// TwinCAT 3 PLC project PLC
// ProgramVersion: 3.1.4024.0
// libraries:
//   SPT Base Types, * (Beckhoff Automation LLC)
//   SPT Components, * (Beckhoff Automation LLC)
//   SPT Event Logger, * (Beckhoff Automation LLC)
//   SPT Motion Control, * (Beckhoff Automation LLC)
//   SPT Utilities, * (Beckhoff Automation LLC)
//   Tc2_MC2, * (Beckhoff Automation GmbH)
//   Tc2_MC2_Drive, * (Beckhoff Automation GmbH)
//   Tc2_NCI, * (Beckhoff Automation GmbH)
//   Tc2_PlcInterpolation, * (Beckhoff Automation GmbH)
//   Tc2_Standard, * (Beckhoff Automation GmbH)
//   Tc2_System, * (Beckhoff Automation GmbH)
//   Tc2_Utilities, * (Beckhoff Automation GmbH)
//   Tc3_EventLogger, * (Beckhoff Automation GmbH)
//   Tc3_Module, * (Beckhoff Automation GmbH)
//   Tc3_PackML_V2, * (Beckhoff Automation GmbH)
//   TcUnit, * (www.tcunit.org)
//   VisuDialogs, * (System)
// project tree:
//   DUTs/ ST_Recipe_Limits.TcDUT, ST_LimitInfo.TcDUT, E_CutDirection.TcDUT, E_PMLStateForHMI.TcTLEO, ST_Machine_HMI.TcDUT, ST_Machine_Status.TcDUT
//   GVLs/ GVL_HMI.TcGVL, GVL_Safety.TcGVL, IO.TcGVL
//   / PlcTask.TcTTO, SafetyTask.TcTTO, Visualization Manager.TcVMO (not stored), VISU_TASK.TcTTO
//   POUs/Builder/ E_ExecutionRoute.TcDUT, I_GeometryWriter.TcIO, FB_RecipeBase.TcPOU, FB_RecipeFactory.TcPOU, I_RecipeBuilder.TcIO, ST_CutSegment.TcDUT, ST_PointXY.TcDUT (not stored), ST_RecipeBuilder_Config.TcDUT, ST_RecipeBuilder_HMI.TcDUT
//   POUs/Builder/Recipes/ FB_FeedMeina2_1000x1000_Circles.TcPOU, FB_FeedMeina2_2000x500.TcPOU, FB_FeedMeina2_750x750.TcPOU, FB_FeedMeina2_750x750_Circles.TcPOU, FB_FeedMeina2_1000x1000.TcPOU, FB_FeedMeina2_500x500.TcPOU, FB_FeedMeina2_500x500_Circles.TcPOU, FB_FeedRoundedRectangle.TcPOU, FB_FeedCircle.TcPOU, FB_FeedMeina2_2000x1000.TcPOU, FB_FeedMeina2_Samples.TcPOU, FB_PTPArona.TcPOU, FB_NCICircle.TcPOU, FB_PTPRectangle.TcPOU, FB_PTPBorgoFlaps.TcPOU, FB_PTPBorgoWings.TcPOU
//   POUs/Components/ FB_Cylinder.TcPOU, I_Cylinder.TcIO, FB_NciChannel.TcPOU, FB_NciChannelTangential.TcPOU, ST_Cylinder_Command.TcDUT, ST_Cylinder_Config.TcDUT, ST_Cylinder_HMI.TcDUT, ST_Cylinder_Status.TcDUT
//   POUs/Components/I_Channel/ ST_NciAxisIds.TcDUT, I_NciChannelBase.TcIO, I_NciChannel_FeedTable.TcIO, I_NciChannel_GCode.TcIO
//   POUs/Executor/ FB_Exec_Pneumatic_PTP.TcPOU, FB_Exec_Drill_PTP.TcPOU, FB_Exec_Tangential_FeedTable.TcPOU, FB_Exec_Spindle_PTP.TcPOU, I_BB8Specification.TcIO, FB_ExecutorBase.TcPOU, I_MachiningExecutor.TcIO, FB_Exec_Spindle_GCodeXYZ.TcPOU
//   POUs/GantryXYZ/ E_MachineProfile.TcDUT, E_RecipeID.TcDUT, ST_AxisProfile.TcDUT, ST_GantryXYZ_Limits.TcDUT, FB_GantryXYZ.TcPOU, I_GantryConfigProvider.TcIO, ST_GantryXYZ_Command.TcDUT, ST_GantryXYZ_Config.TcDUT, ST_GantryXYZ_HMI.TcDUT, ST_GantryXYZ_Status.TcDUT (not stored)
//   POUs/GantryXYZ/HomingStrategies/ FB_Homing_Base.TcPOU, FB_Homing_CustomPLC.TcPOU, FB_Homing_Direct.TcPOU, FB_Homing_StandardNC.TcPOU, I_HomingStrategy.TcIO
//   POUs/ FB_Machine.TcPOU, FB_PersistentDataManager.TcPOU, GlobalTextList.TcGTLO, MAIN.TcPOU, SAFETY.TcPOU, TESTS.TcPOU
//   POUs/TESTS/ FB_Cylinder_Test.TcPOU, FB_ExecutorNCITable_Test.TcPOU, FB_ExecutorGCode_Test.TcPOU, FB_FeedBuilderRoundedRect_Test.TcPOU, FB_NciChannelTangential_Test.TcPOU, FB_NciChannel_Test.TcPOU, FB_GantryXYZ_Test.TcPOU, FB_ExecutorCut_Test.TcPOU, FB_ExecutorGrooveXY_Test.TcPOU, FB_RecipeBuilder_Test.TcPOU, FB_RecipeFactory_Test.TcPOU, FB_Exec_Drill_PTP_Test.TcPOU
//   POUs/TESTS/Mocks/ FB_MockAxis.TcPOU, FB_MockRecipe_Drill.TcPOU, FB_MockGeometryWriter.TcPOU, FB_MockNciChannelFeedTable.TcPOU, FB_MockNciChannel.TcPOU, FB_MockCylinder.TcPOU, FB_MockConfigProvider.TcPOU
//   VISUs/Modes/ProductionMode/ V_Builders.TcVIS, V_Meina2_Samples.TcVIS, V_ProductionArona.TcVIS, V_ProductionFeedCircle.TcVIS, V_ProductionMeina2_5Squares.TcVIS, V_ProductionMeina2_5Circles.TcVIS, V_ProductionMeina2_3Squares.TcVIS, V_ProductionMeina2_3Circles.TcVIS, V_ProductionMeina2_2Squares.TcVIS, V_ProductionMeina2_2Circles.TcVIS, V_ProductionMeina2_2Rectangles.TcVIS, V_ProductionRoundRectangle.TcVIS, V_ProductionRectangle.TcVIS, V_ProductionNCICircle.TcVIS, V_ProductionBorgoFlaps.TcVIS, V_ProductionBorgoWings.TcVIS, V_Meina2_2000x1000.TcVIS, V_ProductionWelcome.TcVIS
//   VISUs/Modes/ V_MaintenanceMode.TcVIS, V_ManualMode.TcVIS, V_ProductionMode.TcVIS
//   VISUs/ V_InfoMenu.TcVIS, V_MainMenu.TcVIS, V_Main.TcVIS
// real-time tasks:
//   TASK PlcTask: cycle T#10ms, priority 20, ADS port 350
//   TASK SafetyTask: cycle T#10ms, priority 21, ADS port 351
//   TASK VISU_TASK: cycle T#200000us, priority 30, ADS port 352
// motion (NC):
//   TASK NC-Task 1 SAF: cycle T#2ms, priority 4, ADS port 501
//   TASK NC-Task 1 SVB: cycle T#10ms, priority 8, ADS port 511
//   AXIS Test Axis X (id 5)
//     OtherSettings: AllowMotionCmdToSlave=true
//     encoder EncType=1
//       Inc: RefSoftSyncMask=#x0000ffff
//     drive DrvType=5
//       Analog: TorqueSetpointScale=10, ScaleFactorActTorque=0.1
//       TimeComp: TaskDelayCycles=1
//     controller CtrType=1
//       CtrPara: PriorControlFactor=1
//         Observer: BandWidth=20
//   AXIS Test Axis Y (id 6)
//     OtherSettings: AllowMotionCmdToSlave=true
//     encoder EncType=1
//     drive DrvType=5
//       Analog: TorqueSetpointScale=10, ScaleFactorActTorque=0.1
//       TimeComp: TaskDelayCycles=1
//     controller CtrType=1
//       CtrPara: PriorControlFactor=1
//         Observer: BandWidth=20
//   AXIS Test Axis Z (id 7)
//     OtherSettings: AllowMotionCmdToSlave=true
//     encoder EncType=1
//     drive DrvType=5
//       Analog: TorqueSetpointScale=10, ScaleFactorActTorque=0.1
//       TimeComp: TaskDelayCycles=1
//     controller CtrType=1
//       CtrPara: PriorControlFactor=1
//         Observer: BandWidth=20
//   AXIS Test Axis Q (id 8)
//     OtherSettings: AllowMotionCmdToSlave=true
//     encoder EncType=1
//     drive DrvType=5
//       Analog: TorqueSetpointScale=10, ScaleFactorActTorque=0.1
//       TimeComp: TaskDelayCycles=1
//     controller CtrType=1
//       CtrPara: PriorControlFactor=1
//         Observer: BandWidth=20
//   AXIS Axis Q (id 1)
//     General: UnitName=°
//     Dynamic: Acceleration=15000, Deceleration=15000, Jerk=45000
//     Velo: RefSearch=720, RefSync=90, SlowManual=30, FastManual=180, Fast=10738.39, Maximum=10738.4
//     TargetPosControl: Range=0.1
//     BacklashCompensation: Range=0.2
//     OtherSettings: AllowMotionCmdToSlave=true, PulseDistancePos=9, PulseDistanceNeg=9
//     encoder EncType=19
//       EncPara: ScaleFactorNumerator=360, ScaleFactorDenominator=3145728, MaxCount=#xffffffff
//         SoftEndMinControl: Range=-300
//         SoftEndMaxControl: Range=300
//     drive DrvType=16
//       DrvPara: MaxCount=#xffffffff, DriveControlDWord=#x00020100
//         Analog: VeloReferenz=11812.229, VeloScale=32, TorqueSetpointScale=10, ScaleFactorActTorque=0.1
//         TimeComp: TaskDelayCycles=1
//     controller CtrType=1
//       CtrPara: PriorControlFactor=1
//         PosDiffControl: Range=40
//         Observer: BandWidth=20
//   AXIS Axis Y (id 2)
//     Dynamic: Acceleration=100, Deceleration=100, Jerk=200
//     Velo: RefSearch=50, RefSync=10, SlowManual=5, FastManual=80, Fast=429.536, Maximum=429.536
//     TargetPosControl: Range=0.1
//     BacklashCompensation: Range=0.1
//     OtherSettings: AllowMotionCmdToSlave=true
//     encoder EncType=19
//       EncPara: ScaleFactorNumerator=4.8, ScaleFactorDenominator=1048576, MaxCount=#xffffffff
//         SoftEndMinControl: Enable=true, Range=-3000
//         SoftEndMaxControl: Enable=true, Range=3000
//         Inc: RefSearchInverse=true, RefSyncInverse=false, RefMode=1
//     drive DrvType=16
//       DrvPara: MaxCount=#xffffffff, DriveControlDWord=#x00020100
//         Analog: VeloReferenz=472.4896, VeloScale=32, TorqueSetpointScale=10, ScaleFactorActTorque=0.1
//         TimeComp: TaskDelayCycles=1
//     controller CtrType=1
//       CtrPara: PriorControlFactor=1
//         Observer: BandWidth=20
//   AXIS Axis Z (id 9)
//     Dynamic: AccelerationMaximum=1200, DecelerationMaximum=1200, Acceleration=20, Deceleration=20, Jerk=80
//     Velo: RefSearch=5, RefSync=2, SlowManual=5, FastManual=10, Maximum=20
//     TargetPosControl: Range=0.1
//     BacklashCompensation: Range=0.1
//     OtherSettings: AllowMotionCmdToSlave=true
//     encoder EncType=4
//       EncPara: ScaleFactorNumerator=2, ScaleFactorDenominator=12800, Inverse=true, MaxCount=#xffffffff
//         Inc: RefPosition=31, RefMode=1
//     drive DrvType=24
//       DrvPara: Inverse=true
//         Analog: VeloReferenz=20, TorqueSetpointScale=10, ScaleFactorActTorque=0.1
//         TimeComp: TaskDelayCycles=1
//     controller CtrType=1
//       CtrPara: PriorControlFactor=1
//         PosDiffControl: Range=2
//         Observer: BandWidth=20
//   AXIS Axis X (id 3)
//     Dynamic: Acceleration=100, Deceleration=100, Jerk=200
//     Velo: RefSearch=50, RefSync=10, SlowManual=5, FastManual=80, Fast=536.92, Maximum=536.92
//     TargetPosControl: Range=0.1
//     BacklashCompensation: Range=0.067
//     OtherSettings: AllowMotionCmdToSlave=true
//     encoder EncType=19
//       EncPara: ScaleFactorNumerator=6, ScaleFactorDenominator=1048576, MaxCount=#xffffffff
//         SoftEndMinControl: Enable=true, Range=-2000
//         SoftEndMaxControl: Enable=true, Range=2000
//         Inc: RefSearchInverse=true, RefSyncInverse=false, RefMode=1
//     drive DrvType=16
//       DrvPara: MaxCount=#xffffffff, DriveControlDWord=#x00020100
//         Analog: VeloReferenz=590.612, VeloScale=32, TorqueSetpointScale=10, ScaleFactorActTorque=0.1
//         TimeComp: TaskDelayCycles=1
//     controller CtrType=1
//       CtrPara: PriorControlFactor=1
//         Observer: BandWidth=20
// I/O:
//   DEVICE Device 3 (EtherCAT), AmsNetId 0.0.0.0.4.1
//     Term 1 (EK1100) [EK1100 EtherCAT Coupler (2A E-Bus)]
//       Term 2 (EL1008) [EL1008 8Ch. Dig. Input 24V, 3ms]
//       Term 3 (EL1008) [EL1008 8Ch. Dig. Input 24V, 3ms]
//       Term 4 (EL2008) [EL2008 8Ch. Dig. Output 24V, 0.5A]
//       Term 5 (EL7221-9014) [EL7221-9014 1Ch. MDP742 Servo motor output stage with OCT (50V, 8A RMS) and STO input]
//         startup 32786:19 := 0000 // DRV Brake Settings / Emergency application timeout
//         startup 32784:51 := 0A00 // DRV Amplifier Settings / Stand still window
//         startup 32785:27 := 01150000 // DRV Motor Settings / Motor speed limitation
//         startup 28688:11 := E803 // DRV Outputs / Torque limitation
//         startup 32784:19 := 5300 // DRV Amplifier Settings / Current loop proportional gain
//         startup 32784:18 := 0500 // DRV Amplifier Settings / Current loop integral time
//         startup 32784:21 := 1F010000 // DRV Amplifier Settings / Velocity loop proportional gain
//         startup 32784:20 := 96000000 // DRV Amplifier Settings / Velocity loop integral time
//         startup 32768:1 := 00 // FB Settings / Invert feedback direction
//       Term 6 (EL7221-9014) [EL7221-9014 1Ch. MDP742 Servo motor output stage with OCT (50V, 8A RMS) and STO input]
//         startup 32785:27 := 01150000 // DRV Motor Settings / Motor speed limitation
//         startup 28688:11 := E803 // DRV Outputs / Torque limitation
//         startup 32784:19 := 5300 // DRV Amplifier Settings / Current loop proportional gain
//         startup 32784:18 := 0500 // DRV Amplifier Settings / Current loop integral time
//         startup 32784:21 := E0000000 // DRV Amplifier Settings / Velocity loop proportional gain
//         startup 32784:20 := 96000000 // DRV Amplifier Settings / Velocity loop integral time
//         startup 32768:1 := 00 // FB Settings / Invert feedback direction
//       Term 7 (EL7221-9014) [EL7221-9014 1Ch. MDP742 Servo motor output stage with OCT (50V, 8A RMS) and STO input]
//         startup 32785:27 := 01150000 // DRV Motor Settings / Motor speed limitation
//         startup 28688:11 := E803 // DRV Outputs / Torque limitation
//         startup 32784:19 := 5300 // DRV Amplifier Settings / Current loop proportional gain
//         startup 32784:18 := 0500 // DRV Amplifier Settings / Current loop integral time
//         startup 32784:21 := E0000000 // DRV Amplifier Settings / Velocity loop proportional gain
//         startup 32784:20 := 96000000 // DRV Amplifier Settings / Velocity loop integral time
//         startup 32768:1 := 00 // FB Settings / Invert feedback direction
//       Term 20 (EL7037) [EL7037 1Ch. Stepper motor output stage (24V, 1.5A)]
//       Term 8 (EL6900) [EL6900, TwinSAFE PLC]
//       Term 9 (EL1904) [EL1904, 4 Ch. Safety Input 24V, TwinSAFE]
//         modules: Module 1 (FSOES)
//       Term 10 (EL2904) [EL2904, 4 Ch. Safety Output 24V, 0.5A, TwinSAFE]
//         modules: Module 1 (FSOES), Module 2 (DO)
//       Term 11 (EL2622) [EL2622 2Ch. Relay Output, NO (230V AC / 30V DC)]
//       Term 12 (EL9011) [EL9011 End Terminal]
// variable links:
//   Device 3 (EtherCAT) <-> Device 3 (EtherCAT)/Term 1 (EK1100)/Term 8 (EL6900)
//     Term 1 (EK1100)/Term 10 (EL2904)/Module 1 (FSOES)/RxPDO/FSOE <-> ConnectionInputs/TwinSafeGroup1.Term 10 (EL2904) - Module 1 (FSOES)_3 TxPDO
//     Term 1 (EK1100)/Term 9 (EL1904)/Module 1 (FSOES)/RxPDO/FSOE <-> ConnectionInputs/TwinSafeGroup1.Term 9 (EL1904) - Module 1 (FSOES)_2 TxPDO
//     Term 1 (EK1100)/Term 10 (EL2904)/Module 1 (FSOES)/TxPDO/FSOE <-> ConnectionOutputs/TwinSafeGroup1.Term 10 (EL2904) - Module 1 (FSOES)_3 RxPDO
//     Term 1 (EK1100)/Term 9 (EL1904)/Module 1 (FSOES)/TxPDO/FSOE <-> ConnectionOutputs/TwinSafeGroup1.Term 9 (EL1904) - Module 1 (FSOES)_2 RxPDO
//   NC-Task 1 SAF/Axes/Axis Q <-> Device 3 (EtherCAT)/Term 1 (EK1100)/Term 5 (EL7221-9014)
//     Drive/Inputs/In/nDataIn1 <-> DRV Following error actual value/Following error actual value
//     Drive/Inputs/In/nDataIn3[0] <-> DRV Torque actual value/Torque actual value
//     Drive/Inputs/In/nDcOutputTime <-> InfoData/DcOutputShift
//     Drive/Inputs/In/nState1 <-> DRV Statusword/Statusword
//     Drive/Inputs/In/nState2 <-> DRV Statusword/Statusword @bit 8
//     Drive/Inputs/In/nState4 @bit 1 <-> WcState/InputToggle
//     Drive/Inputs/In/nState4 <-> WcState/WcState
//     Drive/Outputs/Out/nCtrl1 <-> DRV Controlword/Controlword
//     Drive/Outputs/Out/nCtrl2 <-> DRV Controlword/Controlword @bit 8
//     Drive/Outputs/Out/nDataOut1 <-> DRV Target position/Target position
//     Drive/Outputs/Out/nDataOut2 <-> DRV Target velocity/Target velocity
//     Enc/Inputs/In/nDataIn1 <-> FB Position/Position
//     Enc/Inputs/In/nDcInputTime <-> InfoData/DcInputShift
//     Enc/Inputs/In/nState4 @bit 1 <-> WcState/InputToggle
//     Enc/Inputs/In/nState4 <-> WcState/WcState
//   NC-Task 1 SAF/Axes/Axis X <-> Device 3 (EtherCAT)/Term 1 (EK1100)/Term 7 (EL7221-9014)
//     Drive/Inputs/In/nDataIn1 <-> DRV Following error actual value/Following error actual value
//     Drive/Inputs/In/nDataIn3[0] <-> DRV Torque actual value/Torque actual value
//     Drive/Inputs/In/nDcOutputTime <-> InfoData/DcOutputShift
//     Drive/Inputs/In/nState1 <-> DRV Statusword/Statusword
//     Drive/Inputs/In/nState2 <-> DRV Statusword/Statusword @bit 8
//     Drive/Inputs/In/nState4 @bit 1 <-> WcState/InputToggle
//     Drive/Inputs/In/nState4 <-> WcState/WcState
//     Drive/Outputs/Out/nCtrl1 <-> DRV Controlword/Controlword
//     Drive/Outputs/Out/nCtrl2 <-> DRV Controlword/Controlword @bit 8
//     Drive/Outputs/Out/nDataOut1 <-> DRV Target position/Target position
//     Drive/Outputs/Out/nDataOut2 <-> DRV Target velocity/Target velocity
//     Enc/Inputs/In/nDataIn1 <-> FB Position/Position
//     Enc/Inputs/In/nDcInputTime <-> InfoData/DcInputShift
//     Enc/Inputs/In/nState4 @bit 1 <-> WcState/InputToggle
//     Enc/Inputs/In/nState4 <-> WcState/WcState
//   NC-Task 1 SAF/Axes/Axis Y <-> Device 3 (EtherCAT)/Term 1 (EK1100)/Term 6 (EL7221-9014)
//     Drive/Inputs/In/nDataIn1 <-> DRV Following error actual value/Following error actual value
//     Drive/Inputs/In/nDataIn3[0] <-> DRV Torque actual value/Torque actual value
//     Drive/Inputs/In/nDcOutputTime <-> InfoData/DcOutputShift
//     Drive/Inputs/In/nState1 <-> DRV Statusword/Statusword
//     Drive/Inputs/In/nState2 <-> DRV Statusword/Statusword @bit 8
//     Drive/Inputs/In/nState4 @bit 1 <-> WcState/InputToggle
//     Drive/Inputs/In/nState4 <-> WcState/WcState
//     Drive/Outputs/Out/nCtrl1 <-> DRV Controlword/Controlword
//     Drive/Outputs/Out/nCtrl2 <-> DRV Controlword/Controlword @bit 8
//     Drive/Outputs/Out/nDataOut1 <-> DRV Target position/Target position
//     Drive/Outputs/Out/nDataOut2 <-> DRV Target velocity/Target velocity
//     Enc/Inputs/In/nDataIn1 <-> FB Position/Position
//     Enc/Inputs/In/nDcInputTime <-> InfoData/DcInputShift
//     Enc/Inputs/In/nState4 @bit 1 <-> WcState/InputToggle
//     Enc/Inputs/In/nState4 <-> WcState/WcState
//   NC-Task 1 SAF/Axes/Axis Z <-> Device 3 (EtherCAT)/Term 1 (EK1100)/Term 20 (EL7037)
//     Drive/Inputs/In/nState1 @bit 3 <-> STM Status/Error
//     Drive/Inputs/In/nState1 @bit 7 <-> STM Status/Motor stall
//     Drive/Inputs/In/nState1 @bit 5 <-> STM Status/Moving negative
//     Drive/Inputs/In/nState1 @bit 4 <-> STM Status/Moving positive
//     Drive/Inputs/In/nState1 @bit 1 <-> STM Status/Ready
//     Drive/Inputs/In/nState1 <-> STM Status/Ready to enable
//     Drive/Inputs/In/nState1 @bit 6 <-> STM Status/Torque reduced
//     Drive/Inputs/In/nState1 @bit 2 <-> STM Status/Warning
//     Drive/Inputs/In/nState2 @bit 3 <-> STM Status/Digital input 1
//     Drive/Inputs/In/nState2 @bit 4 <-> STM Status/Digital input 2
//     Drive/Inputs/In/nState2 @bit 5 <-> STM Status/Sync error
//     Drive/Inputs/In/nState2 @bit 7 <-> STM Status/TxPDO Toggle
//     Drive/Inputs/In/nState4 @bit 1 <-> WcState/InputToggle
//     Drive/Inputs/In/nState4 <-> WcState/WcState
//     Drive/Outputs/Out/nCtrl1 <-> STM Control/Enable
//     Drive/Outputs/Out/nCtrl1 @bit 2 <-> STM Control/Reduce torque
//     Drive/Outputs/Out/nCtrl1 @bit 1 <-> STM Control/Reset
//     Drive/Outputs/Out/nCtrl2 @bit 3 <-> STM Control/Digital output 1
//     Drive/Outputs/Out/nDataOut1 <-> STM Position/Position
//     Enc/Inputs/In/nDataIn1 <-> ENC Status/Counter value
//     Enc/Inputs/In/nDataIn2 <-> ENC Status/Latch value
//     Enc/Inputs/In/nState1 @bit 4 <-> ENC Status/Counter overflow
//     Enc/Inputs/In/nState1 @bit 3 <-> ENC Status/Counter underflow
//     Enc/Inputs/In/nState1 @bit 7 <-> ENC Status/Extrapolation stall
//     Enc/Inputs/In/nState1 <-> ENC Status/Latch C valid
//     Enc/Inputs/In/nState1 @bit 1 <-> ENC Status/Latch extern valid
//     Enc/Inputs/In/nState1 @bit 2 <-> ENC Status/Set counter done
//     Enc/Inputs/In/nState2 @bit 4 <-> ENC Status/Status of extern latch
//     Enc/Inputs/In/nState2 <-> ENC Status/Status of input A
//     Enc/Inputs/In/nState2 @bit 1 <-> ENC Status/Status of input B
//     Enc/Inputs/In/nState2 @bit 2 <-> ENC Status/Status of input C
//     Enc/Inputs/In/nState2 @bit 5 <-> ENC Status/Sync error
//     Enc/Inputs/In/nState2 @bit 7 <-> ENC Status/TxPDO Toggle
//     Enc/Inputs/In/nState4 @bit 1 <-> WcState/InputToggle
//     Enc/Inputs/In/nState4 <-> WcState/WcState
//     Enc/Outputs/Out/nCtrl1 <-> ENC Control/Enable latch C
//     Enc/Outputs/Out/nCtrl1 @bit 3 <-> ENC Control/Enable latch extern on negative edge
//     Enc/Outputs/Out/nCtrl1 @bit 1 <-> ENC Control/Enable latch extern on positive edge
//     Enc/Outputs/Out/nCtrl1 @bit 2 <-> ENC Control/Set counter
//     Enc/Outputs/Out/nDataOut1 <-> ENC Control/Set counter value
//   PLC/PLC Instance <-> Device 3 (EtherCAT)/Term 1 (EK1100)/Term 2 (EL1008)
//     PlcTask Inputs/IO.ProximitySensorX <-> Channel 4/Input
//     PlcTask Inputs/IO.ProximitySensorY <-> Channel 5/Input
//     PlcTask Inputs/IO.ProximitySensorZ <-> Channel 6/Input
//     PlcTask Inputs/MAIN.Seedra.GantryXYZ.CylinderCuttingX.Sensor <-> Channel 8/Input
//     PlcTask Inputs/MAIN.Seedra.GantryXYZ.CylinderCuttingY.Sensor <-> Channel 7/Input
//   PLC/PLC Instance <-> Device 3 (EtherCAT)/Term 1 (EK1100)/Term 4 (EL2008)
//     PlcTask Outputs/IO.CoolingEnable <-> Channel 4/Output
//     PlcTask Outputs/IO.SpindleEnable <-> Channel 3/Output
//     PlcTask Outputs/MAIN.Seedra.GantryXYZ.CylinderCuttingX.Valve <-> Channel 6/Output
//     PlcTask Outputs/MAIN.Seedra.GantryXYZ.CylinderCuttingY.Valve <-> Channel 5/Output
//   PLC/PLC Instance <-> Device 3 (EtherCAT)/Term 1 (EK1100)/Term 8 (EL6900)
//     PlcTask Inputs/GVL_Safety.ComError <-> StandardInputs/TwinSafeGroup1.GVL_Safety.ComError_8
//     PlcTask Inputs/GVL_Safety.FBError <-> StandardInputs/TwinSafeGroup1.GVL_Safety.FBError_6
//     PlcTask Inputs/GVL_Safety.SafeError <-> StandardInputs/TwinSafeGroup1.GVL_Safety.SafeError_7
//     PlcTask Inputs/GVL_Safety.SafetyPermission <-> StandardInputs/TwinSafeGroup1.GVL_Safety.SafetyPermission_11
//     PlcTask Outputs/GVL_Safety.ErrorAck <-> StandardOutputs/TwinSafeGroup1.GVL_Safety.ErrorAck_1
//     PlcTask Outputs/GVL_Safety.RestartFBs <-> StandardOutputs/TwinSafeGroup1.GVL_Safety.RestartFBs_5
//     PlcTask Outputs/GVL_Safety.RunStop <-> StandardOutputs/TwinSafeGroup1.GVL_Safety.RunStop_4
//   PLC/PLC Instance <-> Device 3 (EtherCAT)/Term 1 (EK1100)/Term 9 (EL1904)
//     PlcTask Inputs/GVL_Safety.eStopButton <-> Module 1 (FSOES)/TxPDO/FSOE/InputChannel1
//   PLC/PLC Instance <-> NC-Task 1 SAF/Axes/Axis Q
//     PlcTask Inputs/MAIN.Seedra.GantryXYZ.AxisQ.BasicAxis._Axis.NcToPlc <-> Outputs/ToPlc
//     PlcTask Outputs/MAIN.Seedra.GantryXYZ.AxisQ.BasicAxis._Axis.PlcToNc <-> Inputs/FromPlc
//   PLC/PLC Instance <-> NC-Task 1 SAF/Axes/Axis X
//     PlcTask Inputs/MAIN.Seedra.GantryXYZ.AxisX.BasicAxis._Axis.NcToPlc <-> Outputs/ToPlc
//     PlcTask Outputs/MAIN.Seedra.GantryXYZ.AxisX.BasicAxis._Axis.PlcToNc <-> Inputs/FromPlc
//   PLC/PLC Instance <-> NC-Task 1 SAF/Axes/Axis Y
//     PlcTask Inputs/MAIN.Seedra.GantryXYZ.AxisY.BasicAxis._Axis.NcToPlc <-> Outputs/ToPlc
//     PlcTask Outputs/MAIN.Seedra.GantryXYZ.AxisY.BasicAxis._Axis.PlcToNc <-> Inputs/FromPlc
//   PLC/PLC Instance <-> NC-Task 1 SAF/Axes/Axis Z
//     PlcTask Inputs/MAIN.Seedra.GantryXYZ.AxisZ.BasicAxis._Axis.NcToPlc <-> Outputs/ToPlc
//     PlcTask Outputs/MAIN.Seedra.GantryXYZ.AxisZ.BasicAxis._Axis.PlcToNc <-> Inputs/FromPlc
//   PLC/PLC Instance <-> NC-Task 1 SAF/NC-Channel
//     PlcTask Inputs/MAIN.Seedra.GantryXYZ.NciChannel.stNciToPlc <-> Outputs/ToPlc
//     PlcTask Outputs/MAIN.Seedra.GantryXYZ.NciChannel.stPlcToNci <-> Inputs/FromPlc
//   PLC/PLC Instance <-> NC-Task 1 SAF/NC-ChannelTangential
//     PlcTask Inputs/MAIN.Seedra.GantryXYZ.NciChannelTangential.stNciToPlc <-> Outputs/ToPlc
//     PlcTask Outputs/MAIN.Seedra.GantryXYZ.NciChannelTangential.stPlcToNci <-> Inputs/FromPlc

CONFIGURATION PLC
    RESOURCE PLC ON TwinCAT3
        TASK PlcTask(INTERVAL := T#10ms, PRIORITY := 20);
        TASK SafetyTask(INTERVAL := T#10ms, PRIORITY := 21);
        TASK VISU_TASK(INTERVAL := T#200000us, PRIORITY := 30);
        PROGRAM MAIN WITH PlcTask : MAIN;
        PROGRAM SAFETY WITH SafetyTask : SAFETY;
        PROGRAM VisuElems_Visu_Prg WITH VISU_TASK : VisuElems.Visu_Prg;
    END_RESOURCE
END_CONFIGURATION

// ---- DUTs/ST_Recipe_Limits.TcDUT
TYPE ST_Recipe_Limits :
STRUCT
    PanelFrontLength     	: ST_LimitInfo;
    PanelFrontWidth      	: ST_LimitInfo;
    PanelHeight          	: ST_LimitInfo;
    RailHeightCorrection 	: ST_LimitInfo;
	CuttingOverpass 	 	: ST_LimitInfo;
	GroovingOverpass 	 	: ST_LimitInfo;
	RequestedCopiesX 	 	: ST_LimitInfo;
	RequestedCopiesY 	 	: ST_LimitInfo;
	GrooveDepthZ		 	: ST_LimitInfo;
	Radius					: ST_LimitInfo;
	Diameter				: ST_LimitInfo;
END_STRUCT
END_TYPE

// ---- DUTs/ST_LimitInfo.TcDUT
TYPE ST_LimitInfo :
STRUCT
    MinVal : REAL;
    MaxVal : REAL;
END_STRUCT
END_TYPE

// ---- DUTs/E_CutDirection.TcDUT
{attribute 'qualified_only'}
{attribute 'strict'}
TYPE E_CutDirection :
(
    eCutX := 0,
    eCutY := 1
	//add other cutters here 
);
END_TYPE

// ---- DUTs/E_PMLStateForHMI.TcTLEO
TYPE E_PMLStateForHMI : (
        Undefined    := 0,
        Clearing     := 1,
        Stopped      := 2,
        Starting     := 3,
        Idle         := 4,
        Suspended    := 5,
        Execute      := 6,
        Stopping     := 7,
        Aborting     := 8,
        Aborted      := 9,
        Holding      := 10,
        Held         := 11,
        Unholding    := 12,
        Suspending   := 13,
        Unsuspending := 14,
        Resetting    := 15,
        Completing   := 16,
        Complete     := 17
    ) DINT;
END_TYPE

// ---- DUTs/ST_Machine_HMI.TcDUT
TYPE ST_Machine_HMI :
    STRUCT
        //Config  	: ST_Machine_Config;
		Status 		: ST_Machine_Status;
		//Command 	: ST_Machine_Command;
    END_STRUCT
END_TYPE

// ---- DUTs/ST_Machine_Status.TcDUT
TYPE ST_Machine_Status :
    STRUCT
		PackMLState : E_PMLStateForHMI;
    END_STRUCT
END_TYPE

// ---- POUs/Builder/E_ExecutionRoute.TcDUT
{attribute 'qualified_only'}
{attribute 'strict'}
TYPE E_ExecutionRoute :
(
    ePTP,              
    eGCode,          
    eFeedTable    
);
END_TYPE

// ---- POUs/Components/I_Channel/ST_NciAxisIds.TcDUT
TYPE ST_NciAxisIds :
STRUCT
    nX  : UDINT;
    nY  : UDINT;
    nZ  : UDINT;
    nQ1 : UDINT;
    nQ2 : UDINT;
    nQ3 : UDINT;
    nQ4 : UDINT;
    nQ5 : UDINT;
END_STRUCT
END_TYPE

// ---- POUs/Components/ST_Cylinder_Command.TcDUT
TYPE ST_Cylinder_Command :
    STRUCT
        Extend  : BOOL;
        Retract : BOOL;
    END_STRUCT
END_TYPE

// ---- POUs/Components/ST_Cylinder_Config.TcDUT
TYPE ST_Cylinder_Config :
    STRUCT
 	ExtendTime : LREAL := 1;
	RetractTime : LREAL := 1;
    END_STRUCT
END_TYPE

// ---- POUs/Components/ST_Cylinder_HMI.TcDUT
TYPE ST_Cylinder_HMI :
    STRUCT
        Config  : ST_Cylinder_Config;
        Command : ST_Cylinder_Command;
        Status  : ST_Cylinder_Status;
    END_STRUCT
END_TYPE

// ---- POUs/Components/ST_Cylinder_Status.TcDUT
TYPE ST_Cylinder_Status :
    STRUCT
        Extended   : BOOL;
        Retracted  : BOOL;
        Extending  : BOOL;
        Retracting : BOOL;
    END_STRUCT
END_TYPE

// ---- POUs/GantryXYZ/E_MachineProfile.TcDUT
{attribute 'qualified_only'}
{attribute 'strict'}
TYPE E_MachineProfile :
(
    eProduction,    
    eManual         
);
END_TYPE

// ---- POUs/GantryXYZ/E_RecipeID.TcDUT
{attribute 'qualified_only'}
TYPE E_RecipeId :
(
    eNone        						:= 0, 
    ePTPBorgoFlaps  					:= 1,
    ePTPBorgoWings  					:= 2,
    ePTPArona       					:= 3,
	eNCICircle 	 						:= 4,
	ePTPRectangle   					:= 5,
	eFeedRoundedRectangle 				:= 6,
	eFeedCircle  						:= 7,
	eFeedMeina2_2000x1000				:= 8,
	eFeedMeina2_500x500    				:= 9,
    eFeedMeina2_500x500_Circles    		:= 10,
    eFeedMeina2_750x750    				:= 11,
    eFeedMeina2_750x750_Circles    		:= 12,
    eFeedMeina2_1000x1000    			:= 13,
    eFeedMeina2_1000x1000_Circles    	:= 14,
    eFeedMeina2_2000x500 				:= 15,
	eFeedMeina2_Samples					:= 16
) := eNone; 
END_TYPE

// ---- POUs/GantryXYZ/ST_AxisProfile.TcDUT
TYPE ST_AxisProfile :
STRUCT
    Acceleration : LREAL;
    Deceleration : LREAL;
    Jerk         : LREAL;       
    SoftLimitMin : LREAL;
    SoftLimitMax : LREAL;
	Velocity	 : LREAL; //Used only for MC_Direct, We want to use speed and parameters from TwinCat Axis Parameters or directly from methods
END_STRUCT
END_TYPE

// ---- POUs/GantryXYZ/ST_GantryXYZ_Limits.TcDUT
TYPE ST_GantryXYZ_Limits :
STRUCT
    CutterXOffsetX		: ST_LimitInfo;
    CutterXOffsetY		: ST_LimitInfo;
    CutterYOffsetX		: ST_LimitInfo;
    CutterYOffsetY		: ST_LimitInfo;
    CuttingSpeedXY		: ST_LimitInfo;
    CuttingIdleTime		: ST_LimitInfo;
    GroovingSpeedXY		: ST_LimitInfo;
    GroovingSpeedZ		: ST_LimitInfo;
    GroovingIdleTime	: ST_LimitInfo;
    RapidSpeedX			: ST_LimitInfo;
	RapidSpeedY			: ST_LimitInfo;
    RapidSpeedZ			: ST_LimitInfo;
    GlobalOffsetX		: ST_LimitInfo;
	GlobalOffsetY		: ST_LimitInfo;
	GlobalOffsetZ		: ST_LimitInfo; 
    RawBoardX			: ST_LimitInfo; 
    RawBoardY			: ST_LimitInfo; 
	RawBoardZ			: ST_LimitInfo;
	SafeClearanceZ		: ST_LimitInfo;
	RapidSpeedQ 		: ST_LimitInfo; 
END_STRUCT
END_TYPE

// ---- POUs/GantryXYZ/ST_GantryXYZ_Command.TcDUT
TYPE ST_GantryXYZ_Command :
    STRUCT
		ProgramIdRequested : E_RecipeID;
    END_STRUCT
END_TYPE

// ---- POUs/GantryXYZ/ST_GantryXYZ_Config.TcDUT
TYPE ST_GantryXYZ_Config :
STRUCT
    CutterXOffsetX   : REAL;
    CutterXOffsetY   : REAL;
    CutterYOffsetX   : REAL;
    CutterYOffsetY   : REAL;
	CuttingSpeedXY	 : REAL;
    CuttingIdleTime  : REAL;
	GroovingSpeedXY  : REAL;
    GroovingSpeedZ   : REAL;
    GroovingIdleTime : REAL;
    RapidSpeedX      : REAL;
    RapidSpeedY      : REAL;
    RapidSpeedZ      : REAL;
    GlobalOffsetX    : REAL;
    GlobalOffsetY    : REAL;
	GlobalOffsetZ    : REAL; 
    RawBoardX        : REAL; 
    RawBoardY        : REAL;
	RawBoardZ        : REAL;
    SafeClearanceZ   : REAL; 
	AxisQ_SavedPos	 : LREAL;
	RapidSpeedQ		 : REAL; 
END_STRUCT
END_TYPE

// ---- POUs/GantryXYZ/ST_GantryXYZ_HMI.TcDUT
TYPE ST_GantryXYZ_HMI :
    STRUCT
        Config  : ST_GantryXYZ_Config;
		Status 	: ST_GantryXYZ_Status;
		Command 	: ST_GantryXYZ_Command;
		Limits  : ST_GantryXYZ_Limits;
    END_STRUCT
END_TYPE

// ---- POUs/Builder/ST_CutSegment.TcDUT
TYPE ST_CutSegment :
STRUCT
    Start : ST_PointXY;
    Stop  : ST_PointXY;
END_STRUCT
END_TYPE

// ---- POUs/Builder/ST_RecipeBuilder_Config.TcDUT
TYPE ST_RecipeBuilder_Config :
STRUCT
    PanelFrontLength     	: REAL;
    PanelFrontWidth      	: REAL;
    PanelHeight          	: REAL;
    RailHeightCorrection 	: REAL;
    CuttingOverpass      	: REAL;
    GroovingOverpass    	: REAL;
    FillAll             	: BOOL; 
    RequestedCopiesX    	: DINT;
    RequestedCopiesY    	: DINT; 
    IsValid             	: BOOL; 
    GCodePath           	: STRING(255); 
    Radius					: REAL;
	Diameter				: REAL; 
    GrooveDepthZ         	: REAL;
	NciStartX				: REAL;
	NciStartY				: REAL; 
END_STRUCT
END_TYPE

// ---- POUs/Builder/ST_RecipeBuilder_HMI.TcDUT
TYPE ST_RecipeBuilder_HMI :
    STRUCT
        Config  : ST_RecipeBuilder_Config;
		Limits  : ST_Recipe_Limits; 
    END_STRUCT
END_TYPE

// ---- GVLs/GVL_HMI.TcGVL
{attribute 'qualified_only'}
VAR_GLOBAL
		//0 - Production Mode, 1 - Manual Mode, 2 - Maintenance Mode
		MenuToDisplay :INT;
		//0 - will keep MainMenu open, 1- InfoMenu overlay during the production
		PopupToDisplay :INT;		
END_VAR

// ---- GVLs/GVL_Safety.TcGVL
{attribute 'qualified_only'}
VAR_GLOBAL

RunStop AT%Q* :BOOL;	
ErrorAck AT%Q* :BOOL;
RestartFBs AT%Q* :BOOL;

FBError AT%I* :BOOL;
SafeError AT%I* :BOOL;
ComError AT%I* :BOOL;

SafetyPermission AT %I* :BOOL;
SafetyPermissionQ AT %Q* :BOOL;
SafetyPermissionI AT %I* :BOOL;

eStopButton		AT %I* :BOOL;
eStopHMI		:BOOL;



END_VAR

// ---- GVLs/IO.TcGVL
VAR_GLOBAL

//Terminal EL1008
	DI1			AT%I*		:	BOOL;
	DI2			AT%I*		:	BOOL;
	DI3			AT%I*		:	BOOL;
	DI4			AT%I*		:	BOOL;
	DI5			AT%I*		:	BOOL;
	DI6			AT%I*		:	BOOL;
	DI7			AT%I*		:	BOOL;
	DI8			AT%I*		:	BOOL;
	
	
	SpindleEnable 				AT%Q*		:	BOOL;
	CoolingEnable				AT%Q*		:	BOOL; 
	
	ProximitySensorX			AT%I*		:	BOOL;
	ProximitySensorY			AT%I*		:	BOOL;
	ProximitySensorZ			AT%I*		:	BOOL;
	

	
	
END_VAR

// ---- POUs/Builder/I_GeometryWriter.TcIO
INTERFACE I_GeometryWriter

METHOD AddArc : BOOL
VAR_INPUT
    TargetX    : LREAL;
    TargetY    : LREAL;
    CenterX    : LREAL;
    CenterY    : LREAL;
    Velo       : LREAL;
    Clockwise  : BOOL; 
END_VAR
END_METHOD

METHOD AddLine : BOOL
VAR_INPUT
    TargetX : LREAL;
    TargetY : LREAL;
    Velo    : LREAL;
END_VAR
END_METHOD

METHOD AddStartPoint : BOOL
VAR_INPUT
    TargetX : LREAL;
    TargetY : LREAL;
END_VAR
END_METHOD

METHOD Clear : BOOL
VAR_INPUT
END_VAR
END_METHOD

METHOD EnableTangentialFollowing : BOOL
VAR_INPUT
END_VAR
END_METHOD

METHOD EndTable : BOOL
VAR_INPUT
END_VAR
END_METHOD

END_INTERFACE

// ---- POUs/Components/I_Channel/I_NciChannelBase.TcIO
INTERFACE I_NciChannelBase EXTENDS I_ComponentBase

METHOD BuildGroup
END_METHOD

PROPERTY ChannelError : BOOL
GET
END_GET
END_PROPERTY

PROPERTY ChannelErrorId : UDINT
GET
END_GET
END_PROPERTY

PROPERTY IsGrouped : BOOL
GET
END_GET
END_PROPERTY

PROPERTY IsReady : BOOL
GET
END_GET
END_PROPERTY

METHOD ResetChannel
VAR_INPUT
END_VAR
END_METHOD

METHOD Stop
VAR_INPUT
END_VAR
END_METHOD

METHOD Ungroup
VAR_INPUT
END_VAR
END_METHOD

END_INTERFACE

// ---- POUs/Components/I_Channel/I_NciChannel_FeedTable.TcIO
INTERFACE I_NciChannel_FeedTable EXTENDS I_NciChannelBase

PROPERTY IsChannelDone : BOOL
GET
END_GET
END_PROPERTY

PROPERTY IsFeedingDone : BOOL
GET
END_GET
END_PROPERTY

METHOD Start
VAR_INPUT
END_VAR
END_METHOD

METHOD StartFeedTable
VAR_IN_OUT
    stTable : ST_NciFeedGroupTable;
END_VAR
END_METHOD

END_INTERFACE

// ---- POUs/Components/I_Channel/I_NciChannel_GCode.TcIO
INTERFACE I_NciChannel_GCode EXTENDS I_NciChannelBase

PROPERTY IsMoving : BOOL
GET
END_GET
END_PROPERTY

PROPERTY IsProgramLoaded : BOOL
GET
END_GET
END_PROPERTY

METHOD LoadProgram
VAR_INPUT
	sProgramPath : STRING(255);
END_VAR
END_METHOD

METHOD Start
VAR_INPUT
END_VAR
END_METHOD

END_INTERFACE

// ---- POUs/Components/I_Cylinder.TcIO
INTERFACE I_Cylinder

PROPERTY Error : BOOL
GET
END_GET
END_PROPERTY

METHOD Extend
VAR_INPUT
END_VAR
END_METHOD

PROPERTY Extended : BOOL
GET
END_GET
END_PROPERTY

METHOD Retract
VAR_INPUT
END_VAR
END_METHOD

PROPERTY Retracted : BOOL
GET
END_GET
END_PROPERTY

END_INTERFACE

// ---- POUs/Executor/I_BB8Specification.TcIO
INTERFACE I_BB8Specification

PROPERTY AxisQ : I_BasicAxis
GET
END_GET
SET
END_SET
END_PROPERTY

PROPERTY AxisX : I_BasicAxis
GET
END_GET
SET
END_SET
END_PROPERTY

PROPERTY AxisY : I_BasicAxis
GET
END_GET
SET
END_SET
END_PROPERTY

PROPERTY AxisZ : I_BasicAxis
GET
END_GET
SET
END_SET
END_PROPERTY

PROPERTY ConfigProvider : I_GantryConfigProvider
GET
END_GET
SET
END_SET
END_PROPERTY

PROPERTY Cylinder : I_Cylinder
GET
END_GET
SET
END_SET
END_PROPERTY

PROPERTY RecipeBuilder : I_RecipeBuilder
GET
END_GET
SET
END_SET
END_PROPERTY

END_INTERFACE

// ---- POUs/Executor/I_MachiningExecutor.TcIO
INTERFACE I_MachiningExecutor

METHOD Abort
VAR_INPUT
END_VAR
END_METHOD

PROPERTY Busy : BOOL
GET
END_GET
END_PROPERTY

PROPERTY Done : BOOL
GET
END_GET
END_PROPERTY

PROPERTY Error : BOOL
GET
END_GET
END_PROPERTY

PROPERTY ErrorID : UDINT
GET
END_GET
END_PROPERTY

METHOD Execute : BOOL
VAR_INPUT
END_VAR
END_METHOD

END_INTERFACE

// ---- POUs/GantryXYZ/HomingStrategies/I_HomingStrategy.TcIO
INTERFACE I_HomingStrategy EXTENDS I_MotionSequence

END_INTERFACE

// ---- POUs/GantryXYZ/I_GantryConfigProvider.TcIO
INTERFACE I_GantryConfigProvider

PROPERTY Config : ST_GantryXYZ_Config
GET
END_GET
SET
END_SET
END_PROPERTY

END_INTERFACE

// ---- POUs/Builder/I_RecipeBuilder.TcIO
INTERFACE I_RecipeBuilder

PROPERTY ActualCopiesX : DINT
GET
END_GET
END_PROPERTY

PROPERTY ActualCopiesY : DINT
GET
END_GET
END_PROPERTY

METHOD Build : BOOL
END_METHOD

PROPERTY Busy : BOOL
GET
END_GET
SET
END_SET
END_PROPERTY

PROPERTY Config : ST_RecipeBuilder_Config
GET
END_GET
SET
END_SET
END_PROPERTY

PROPERTY ConfigProvider : I_GantryConfigProvider
GET
END_GET
SET
END_SET
END_PROPERTY

PROPERTY CurrentShapeIndex : INT
GET
END_GET
SET
END_SET
END_PROPERTY

PROPERTY Done : BOOL
GET
END_GET
SET
END_SET
END_PROPERTY

PROPERTY Error : BOOL
GET
END_GET
SET
END_SET
END_PROPERTY

PROPERTY ExecutionRoute : E_ExecutionRoute
GET
END_GET
END_PROPERTY

PROPERTY FootprintX : REAL
GET
END_GET
SET
END_SET
END_PROPERTY

PROPERTY FootprintY : REAL
GET
END_GET
SET
END_SET
END_PROPERTY

PROPERTY GeometryWriter : I_GeometryWriter
GET
END_GET
SET
END_SET
END_PROPERTY

PROPERTY HolesDrill : REFERENCE TO ARRAY [1..100] OF ST_PointXY;
GET
END_GET
END_PROPERTY

PROPERTY HolesToDrill : INT
GET
END_GET
END_PROPERTY

PROPERTY Limits : ST_Recipe_Limits
GET
END_GET
END_PROPERTY

PROPERTY MaxCopiesX : DINT
GET
END_GET
END_PROPERTY

PROPERTY MaxCopiesY : DINT
GET
END_GET
END_PROPERTY

PROPERTY SegmentsCutX : REFERENCE TO ARRAY [1..100] OF ST_CutSegment
GET
END_GET
END_PROPERTY

PROPERTY SegmentsCutY : REFERENCE TO ARRAY [1..100] OF ST_CutSegment
GET
END_GET
END_PROPERTY

PROPERTY SegmentsGroove : REFERENCE TO ARRAY [1..100] OF ST_CutSegment
GET
END_GET
END_PROPERTY

PROPERTY SegmentsToCutX : INT
GET
END_GET
END_PROPERTY

PROPERTY SegmentsToCutY : INT
GET
END_GET
END_PROPERTY

PROPERTY SegmentsToGroove : INT
GET
END_GET
END_PROPERTY

PROPERTY ShapesCount : INT
GET
END_GET
END_PROPERTY

PROPERTY ShapeStart : REFERENCE TO ARRAY [1..100] OF ST_PointXY
GET
END_GET
END_PROPERTY

END_INTERFACE

// ---- POUs/MAIN.TcPOU
PROGRAM MAIN

	VAR
		Seedra          : FB_Machine := (Name := 'SeedraMAIN');
		InitComplete    : BOOL;
		RebootSystem	: NT_Reboot;
	END_VAR

CyclicLogic();
//TESTS();

METHOD CyclicLogic
VAR_INPUT
END_VAR
IF NOT InitComplete THEN
    InitComplete := Initialize();
    RETURN;
END_IF

//Machine support HMI & Production Monitor


//Machine Cyclic Logic
Seedra.CyclicLogic();
END_METHOD

METHOD Initialize : BOOL
VAR_INPUT
END_VAR
//Top level machine initialization should happen here, in the main initialization method. Each subsequent "layer" of modules will be named within their respective "parent" intialize method
_AppInfo.KeepOutputsOnBP := TRUE;
Initialize := TRUE;
END_METHOD

END_PROGRAM

// ---- POUs/FB_Machine.TcPOU
FUNCTION_BLOCK FB_Machine EXTENDS FB_PackML_BaseModule // IMPLEMENTS I_ControlsProductionRate
VAR
    // Sub Modules
    GantryXYZ   : FB_GantryXYZ  := (Name := 'Gantry', LogStateChanges := FALSE);

    //Initial List of Components
    ipComponents_Init : ARRAY[1..Parameters_PackML_Base.MAX_NO_OF_COMPONENTS] OF I_ComponentBase := [];

	//Alarms for this module
	MachineAlarms : ARRAY[1..MACHINE_ALARM_COUNT] OF FB_TcAlarm;
	
	
	ConfigManager :FB_PersistentDataManager;
	RecipeFactory : FB_RecipeFactory;
    RecipeConfig_HMI : ST_RecipeBuilder_HMI; 

	Machine_HMI : ST_Machine_HMI;
	
	sSelectedRecipeName : STRING(50);
	aRecipeNames : ARRAY[0..30] OF STRING(50);


END_VAR

VAR CONSTANT
    MACHINE_ALARM_COUNT : INT := 6;
END_VAR


METHOD PROTECTED Clearing
VAR
	i				: UDINT;
	SubModulesReady : BOOL := TRUE;
END_VAR
CASE SequenceState OF
    0:
        NoStateTasksToComplete := FALSE;
        SequenceState          := SequenceState + 10;
    10:
		//Leave Aborted thanks to this
		MachineAlarms[E_Seedra.EmergencyStop].Clear(0, 0);
        SequenceState := SequenceState + 10;
    20:
		IF ResetSafety() THEN
			SequenceState := SequenceState + 10;		
		END_IF	

	30:
		StateTasksComplete := TRUE; 
			 
END_CASE

SUPER^.Clearing();
END_METHOD

METHOD PROTECTED CreateEvents
VAR_INPUT
END_VAR
// Add your event creation here
F_CreateAllEventsInClass(Alarms     := MachineAlarms,
                         ClassSize  := SIZEOF(TC_Events.Seedra),
                         pInitEvent := ADR(TC_EVENTS.Seedra.InitReferenceEvent),
                         Prefix     := Name);
// Super call to base
SUPER^.CreateEvents();
END_METHOD

METHOD CyclicLogic
VAR
    CurrentBuilder : I_RecipeBuilder;
END_VAR
// =========================================================
// 1. INICJALIZACJA
// =========================================================
IF NOT _InitComplete THEN
    _InitComplete := Initialize();
    RETURN;
END_IF

// =========================================================
// 2. LOGIKA BAZOWA (Maszyna Stanów, Submoduły)
// =========================================================
SUPER^.CyclicLogic();

// =========================================================
// 3. OOP ACTIVE CLAMPING & LIMITS (Single Source of Truth)
// =========================================================
// Wyciągamy interfejs programu, który aktualnie jest wybrany na HMI
CurrentBuilder := RecipeFactory.GetBuilder(GantryXYZ.ProgramIdRequested);

// Synchronizujemy dane z HMI TYLKO gdy maszyna NIE produkuje detalu!
// Zapobiega to wyzerowaniu ścieżki GCodePath przez HMI tuż po jej wygenerowaniu.
IF _CurrentState = E_PMLState.ePMLState_Idle OR 
   _CurrentState = E_PMLState.ePMLState_Stopped OR
   _CurrentState = E_PMLState.ePMLState_Aborted THEN

IF CurrentBuilder <> 0 THEN
    // Wrzucamy dane z HMI -> Wyzwala to limity i UpdateNestingLimits() w Builderze!
    // Builder wewnątrz tej metody sam pyta Gantry o GlobalOffset!
    CurrentBuilder.Config := RecipeConfig_HMI.Config;
        
    // Odczyt z powrotem na HMI (aby wyświetlić przeliczone limity sztuk)
    RecipeConfig_HMI.Config := CurrentBuilder.Config;
    RecipeConfig_HMI.Limits := CurrentBuilder.Limits;
ELSE
    IF GantryXYZ.ProgramIdRequested <> E_RecipeID.eNone THEN
        GantryXYZ.ProgramIdRequested := E_RecipeID.eNone;
    END_IF
END_IF

    // =========================================================
    // 4. ZAPIS DO PERSISTENTÓW I FABRYKI 
    // =========================================================
    ConfigManager.GantryConfig := GantryXYZ.Config;
    ConfigManager.Config := RecipeConfig_HMI.Config;
    RecipeFactory.UpdateConfig(RecipeConfig_HMI.Config);

END_IF

// =========================================================
// 5. OBSŁUGA BEZPIECZEŃSTWA (SAFETY)
// =========================================================
IF (GVL_Safety.eStopHMI OR NOT GVL_Safety.eStopButton) AND NOT MachineAlarms[E_Seedra.EmergencyStop].bRaised THEN
    THIS^.ChangeState(E_PMLCommand.ePMLCommand_Abort);
    RaiseAlarmWithStrings(MachineAlarms[E_Seedra.EmergencyStop],'','');
END_IF
END_METHOD

METHOD PROTECTED Execute
CASE _CurrentMode OF

	//=================================PRODUCTION MODE==================================
	E_PMLUnitMode.ePMLUnitMode_Production:
	CASE SequenceState OF
			0:
				NoStateTasksToComplete := FALSE;
				// FABRYKA DAJE NAM ODPOWIEDNI INTERFEJS NA BAZIE WYBORU Z HMI
				GantryXYZ.RecipeBuilder := RecipeFactory.GetBuilder(GantryXYZ.ProgramIdRequested);
				
				IF GantryXYZ.RecipeBuilder <> 0 THEN
					GantryXYZ.ChangeState(E_PMLCommand.ePMLCommand_Start);
					SequenceState := 10; // Ręczne przypisanie konkretnego kroku (bezpieczniejsze)
				ELSE
					// Brak buildera = zły numer programu
					ChangeState(E_PMLCommand.ePMLCommand_Abort);
				END_IF
				
			10: 
                // Czekamy, aż moduł Gantry zamelduje zakończenie obróbki
                IF GantryXYZ.CurrentState = E_PMLState.ePMLState_Complete THEN
                    SequenceState := 20;
                
                // --- DODAJ TEN WARUNEK ---
                ELSIF GantryXYZ.CurrentState = E_PMLState.ePMLState_Aborting OR GantryXYZ.CurrentState = E_PMLState.ePMLState_Aborted THEN
                    // Jeśli submoduł Gantry uległ awarii, wymuś awarię całej maszyny!
                    ChangeState(E_PMLCommand.ePMLCommand_Abort);
                    SequenceState := 999; 
                END_IF  
                    
            20:
                StateTasksComplete := TRUE;
                StateComplete();
                
            999:
                // Martwy krok dla awarii
                ;
				
		END_CASE

	//=================================MAINTENANCE & MANUAL MODE==================================
	E_PMLUnitMode.ePMLUnitMode_Maintenance, E_PMLUnitMode.ePMLUnitMode_Manual:
		;
END_CASE
END_METHOD

//! @summary Provides interlocks for HMI control and updates HMI status information for this module
METHOD PROTECTED HMICommunication

//! @description This method is called cyclically by <c>CyclicLogic()</c>
VAR
// Just to get rid of annoing warring 
CastingHelper : DINT; 
END_VAR

IF GVL_Safety.eStopHMI THEN
	PackMLBaseModule_HMI.Status.Error := TRUE;
	THIS^._Error := TRUE;
END_IF

CastingHelper := _CurrentState;
Machine_HMI.Status.PackMLState := CastingHelper;

aRecipeNames[E_RecipeID.eNone]       					:= '-';
aRecipeNames[E_RecipeID.ePTPBorgoFlaps] 				:= 'Borgo Flaps';
aRecipeNames[E_RecipeID.ePTPBorgoWings] 				:= 'Borgo Wings';
aRecipeNames[E_RecipeID.ePTPArona]      				:= 'Arona';
aRecipeNames[E_RecipeID.eNCICircle]  					:= 'NCI Circle';
aRecipeNames[E_RecipeID.ePTPRectangle]					:= 'Rectangle';
aRecipeNames[E_RecipeID.eFeedRoundedRectangle]			:= 'Rounded Rectangle';
aRecipeNames[E_RecipeID.eFeedCircle]					:= 'Feed Circle';
aRecipeNames[E_RecipeID.eFeedMeina2_2000x1000]			:= 'Meina Rectangle 2000x1000';
aRecipeNames[E_RecipeID.eFeedMeina2_500x500]    		:= 'Meina Mix 500x500';
aRecipeNames[E_RecipeID.eFeedMeina2_500x500_Circles]    := 'Meina Mix Circles 500';
aRecipeNames[E_RecipeID.eFeedMeina2_750x750]    		:= 'Meina Squares 750x750';
aRecipeNames[E_RecipeID.eFeedMeina2_750x750_Circles]   	:= 'Meina Circles 750';
aRecipeNames[E_RecipeID.eFeedMeina2_1000x1000]    		:= 'Meina Squares 1000x1000';
aRecipeNames[E_RecipeID.eFeedMeina2_1000x1000_Circles]  := 'Meina Circles 1000x1000';
aRecipeNames[E_RecipeID.eFeedMeina2_2000x500] 			:= 'Meina Rectangles 2000x500';
aRecipeNames[E_RecipeID.eFeedMeina2_Samples] 			:= 'Meina Samples';


sSelectedRecipeName := aRecipeNames[GantryXYZ.ProgramIdRequested];

SUPER^.HMICommunication();
END_METHOD

METHOD PROTECTED HMIPermissions
//General Mode Based Monitoring and handling of HMI control
CASE _CurrentMode OF
   
 E_PMLUnitMode.ePMLUnitMode_Production:
 		
 		GVL_HMI.MenuToDisplay := 0;
 	
        CASE _CurrentState OF
			
            E_PMLState.ePMLState_Stopped:
				AllowHMIControl(ThisModuleOnly := FALSE);
            E_PMLState.ePMLState_Idle:
				GVL_HMI.MenuToDisplay := 0;
				AllowHMIControl(ThisModuleOnly := FALSE);
            E_PMLState.ePMLState_Suspended:
         		AllowHMIControl(ThisModuleOnly := FALSE);
            E_PMLState.ePMLState_Execute:
				GVL_HMI.PopupToDisplay := 1;
            	AllowHMIControl(ThisModuleOnly := FALSE); 
			  E_PMLState.ePMLState_Aborting:
				GVL_HMI.PopupToDisplay := 0;
				AllowHMIControl(ThisModuleOnly := FALSE); 
            E_PMLState.ePMLState_Aborted:
				GVL_HMI.MenuToDisplay := 0;
                AllowHMIControl(ThisModuleOnly := FALSE); 
            E_PMLState.ePMLState_Held:
                AllowHMIControl(ThisModuleOnly := FALSE); 
            E_PMLState.ePMLState_Complete:
				GVL_HMI.PopupToDisplay := 0;
          		AllowHMIControl(ThisModuleOnly := FALSE); 
				
        END_CASE
		
	E_PMLUnitMode.ePMLUnitMode_Maintenance:
		GVL_HMI.MenuToDisplay := 2;
        AllowHMIControl(ThisModuleOnly := FALSE); 
		
    E_PMLUnitMode.ePMLUnitMode_Manual:
		GVL_HMI.MenuToDisplay := 1;
        AllowHMIControl(ThisModuleOnly := FALSE); 

END_CASE
END_METHOD

METHOD PROTECTED Initialize : BOOL
VAR
    i : UDINT; //Generic iteration value
END_VAR
Initialize := FALSE;
CASE DescendantSequenceState OF
    0:
		RegisterSubmodule(GantryXYZ);

        _LogModeChanges         := FALSE;
        _LogStateChanges        := FALSE;
  
	    DescendantSequenceState := DescendantSequenceState + 10;
    10:
        DescendantSequenceState := DescendantSequenceState + 10;
    20:
        //Copy Mode names
        FOR i := 1 TO 3 DO
            ModeNames[i] := F_UnitModeToString(UDINT_TO_DINT(i));
        END_FOR

        DescendantSequenceState := DescendantSequenceState + 10;
    30:
        // Initialize Safety
		IF NOT GVL_Safety.RunStop THEN
			GVL_Safety.RunStop := TRUE;	
		END_IF
        DescendantSequenceState := DescendantSequenceState + 10;
	
	40: 

		// Przekazanie konfiguracji do Gantry
		GantryXYZ.Config := ConfigManager.GantryConfig;
		
		// Przekazanie konfiguracji z Persistenta do Fabryki ORAZ wstrzyknięcie maszyny (GantryXYZ)
		RecipeFactory.InitializeFactory(Config := ConfigManager.Config, ConfigProvider := GantryXYZ);
	
		// Przekazanie konfiguracji z Persistenta do HMI (żeby po restarcie na ekranie były dobre wartości)
		RecipeConfig_HMI.Config := ConfigManager.Config;
		
		// =================================================================================
		// DOMYŚLNE LIMITY FIZYCZNE MASZYNY (Zabezpieczenie Numpadów na ekranie powitalnym)
		// =================================================================================
//		RecipeConfig_HMI.Limits.PanelFrontLength.MinVal 	:= 12.0;     RecipeConfig_HMI.Limits.PanelFrontLength.MaxVal 	:= 1234.0;
//		RecipeConfig_HMI.Limits.PanelFrontWidth.MinVal  	:= 12.0;     RecipeConfig_HMI.Limits.PanelFrontWidth.MaxVal  	:= 1234.0;
//		RecipeConfig_HMI.Limits.PanelHeight.MinVal      	:= 12.0;     RecipeConfig_HMI.Limits.PanelHeight.MaxVal      	:= 1234.0;
//		RecipeConfig_HMI.Limits.RailHeightCorrection.MinVal := 12.0; 	 RecipeConfig_HMI.Limits.RailHeightCorrection.MaxVal := 1234.0;
		RecipeConfig_HMI.Limits.CuttingOverpass.MinVal 		:= 0.0;      RecipeConfig_HMI.Limits.CuttingOverpass.MaxVal 	:= 50.0;
		RecipeConfig_HMI.Limits.GroovingOverpass.MinVal 	:= 0.0;      RecipeConfig_HMI.Limits.GroovingOverpass.MaxVal 	:= 50.0;
		RecipeConfig_HMI.Limits.GrooveDepthZ.MinVal := 0.0;
		RecipeConfig_HMI.Limits.GrooveDepthZ.MaxVal := 100.0;
		
		IF RecipeConfig_HMI.Config.RequestedCopiesX < 1 THEN RecipeConfig_HMI.Config.RequestedCopiesX := 1; END_IF
		IF RecipeConfig_HMI.Config.RequestedCopiesY < 1 THEN RecipeConfig_HMI.Config.RequestedCopiesY := 1; END_IF
		
		
		// Przekazanie konfiguracji z Persistenta do Fabryki (Fabryka rozda to builderom)
		RecipeFactory.UpdateConfig(ConfigManager.Config);
	
		DescendantSequenceState := DescendantSequenceState + 10;
		
    50:
        //Call the Super
        IF SUPER^.Initialize() THEN
            DescendantSequenceState := DescendantSequenceState + 10;
        END_IF

    60:
        Initialize := TRUE;
END_CASE
END_METHOD

METHOD ResetSafety : BOOL
VAR_INST
	Step : INT ;	
	SafetyTimer :TON;
	SafetyTimerTrigger :R_TRIG;
END_VAR
//auto resetting timer, a start condition is an end condition
SafetyTimer(IN:= Step > 0 AND NOT SafetyTimer.Q, PT:= T#500MS);

CASE Step OF
		
		0:  // Reset group or waits
			ResetSafety:= FALSE;
			//Trace('Timer Initialize');
			Step := Step + 10;
			
		10: //If necessary reset group
		
			GVL_Safety.ErrorAck := (GVL_Safety.ComError OR GVL_Safety.FBError); 
		
			IF GVL_Safety.ErrorAck OR SafetyTimer.Q THEN 
				Step := Step + 10;
			END_IF

		20: //Wait for the signal propagation
			IF SafetyTimer.Q THEN
				GVL_Safety.ErrorAck := FALSE;
				Step := Step + 10;
			END_IF
		
		30: //Check FB errors
			IF GVL_Safety.FBError OR (NOT GVL_Safety.SafetyPermission) THEN
				GVL_Safety.RestartFBs := TRUE;
			END_IF
			
			Step := Step + 10;
			
		40: //Wait for the signal propagation
		
			IF SafetyTimer.Q THEN
				GVL_Safety.RestartFBs := FALSE;
				Step := Step + 10;
			END_IF	
			
		50: //Wait for the signal propagation
			
			
		IF SafetyTimer.Q THEN
				
			
				IF GVL_Safety.SafetyPermission AND 
					NOT (GVL_Safety.ComError OR GVL_Safety.FBError OR GVL_Safety.SafeError) 
				
					THEN
						Step := 0;
						ResetSafety := TRUE;
					ELSE
						Step := 0;
						ResetSafety := FALSE;
				END_IF
			
			END_IF
		
		ELSE
		
		Step := 0;	

END_CASE
END_METHOD

METHOD PROTECTED Resetting
VAR
	i				: UDINT;
	SubModulesReady : BOOL := TRUE;
END_VAR
CASE _CurrentMode OF

	//=================================PRODUCTION MODE==================================
	E_PMLUnitMode.ePMLUnitMode_Production:
		CASE SequenceState OF
			0:
				NoStateTasksToComplete := FALSE;

				GantryXYZ.ChangeState(E_PMLCommand.ePMLCommand_Reset);
				
				SequenceState := SequenceState + 10;
					
			10:
				StateTasksComplete := TRUE;
				
			
		END_CASE

	//=================================MAINTENANCE & MANUAL MODE==================================
	E_PMLUnitMode.ePMLUnitMode_Maintenance, E_PMLUnitMode.ePMLUnitMode_Manual:
;
END_CASE

SUPER^.Resetting();
END_METHOD

//! @summary This method monitors <b>submodules</b> within this PackML module and initiates fault responses as required
METHOD PROTECTED SubModuleMonitor : BOOL
VAR
	AlarmResponses : ARRAY[0..4] OF E_AlarmResponse; //Temporary response array	
	i			   : UDINT;
END_VAR

//! @description This method is called cyclically by <c>CyclicLogic()</c>
// Check the sub Modules for Alarm Severity
SUPER^.SubModuleMonitor();

//Check the alarms at the machine level
_CurrentAlarmSeverity := F_GetMaxSeverityRaised(Alarms := MachineAlarms, CurrentSeverity := _CurrentAlarmSeverity);

//Check the severity of the machine level alarms
IF _CurrentState <> E_PMLState.ePMLState_Aborted AND _CurrentState <> E_PMLState.ePMLState_Aborting AND _CurrentState <> E_PMLState.ePMLState_Clearing  AND
   _CurrentState <> E_PMLState.ePMLState_Stopped AND _CurrentState <> E_PMLState.ePMLState_Stopping THEN
    AlarmResponses := _ParentFaultResponseDefinitions;
    CASE AlarmResponses[CurrentAlarmSeverity] OF
        E_AlarmResponse.Abort_ImmediateError:
            AbortImmediateError(Name, TRUE);
        E_AlarmResponse.Abort_Immediate:
            AbortImmediate();
        E_AlarmResponse.Stop_Immediate:
            StopImmediate();
        E_AlarmResponse.Stop_Controlled:
            StopControlled();
        E_AlarmResponse.Hold_Immediate:
            HoldImmediate();
        E_AlarmResponse.Suspend_Immediate:
            SuspendImmediate();
        E_AlarmResponse.Suspend_Controlled:
            SuspendControlled();
        E_AlarmResponse.NoResponse:
            ;
    END_CASE
ELSIF _CurrentState = E_PMLState.ePMLState_Stopped OR _CurrentState = E_PMLState.ePMLState_Stopping THEN
    AlarmResponses := _ParentFaultResponseDefinitions;
    CASE AlarmResponses[CurrentAlarmSeverity] OF
        E_AlarmResponse.Abort_ImmediateError:
            AbortImmediateError(Name, TRUE);
        E_AlarmResponse.Abort_Immediate:
            AbortImmediate();
        E_AlarmResponse.NoResponse:
            ;
    END_CASE
END_IF
END_METHOD

END_FUNCTION_BLOCK

// ---- POUs/GantryXYZ/FB_GantryXYZ.TcPOU
{attribute 'conditionalshow'}
FUNCTION_BLOCK FB_GantryXYZ EXTENDS FB_PackML_BaseModule IMPLEMENTS I_GantryConfigProvider
VAR
	
	fbHomeMcQ           : MC_Home;
    // =========================================================
    //  DEPENDENCIES & SUB-MODULES
    // =========================================================
    _RecipeBuilder      : I_RecipeBuilder;
    ipSubModules_Init   : ARRAY[1..Parameters_PackML_Base.MAX_NO_OF_SUBMODULES] OF I_PackML_BaseModule := [];

	ExecutorCutX 		: FB_Exec_Pneumatic_PTP;
	ExecutorCutY 		: FB_Exec_Pneumatic_PTP;	
	ExecutorGrooveXY	: FB_Exec_Spindle_PTP;
	ExecutorDrill 		: FB_Exec_Drill_PTP;
	ExecTangentialFeed	: FB_Exec_Tangential_FeedTable;
	
	ExecutorNCI 		: FB_Exec_Spindle_GCodeXYZ;
	
	_Limits : ST_GantryXYZ_Limits;


    // =========================================================
    //  HMI & COMMANDS
    // =========================================================
    GantryXYZ_HMI       : ST_GantryXYZ_HMI;
    _ProgramIdRequested : E_RecipeID;

    // =========================================================
    //  COMPONENTS (AXES & CYLINDERS)
    // =========================================================
    AxisX               : FB_Component_BasicAxis := (Name := 'AxisX');
    AxisY               : FB_Component_BasicAxis := (Name := 'AxisY');
    AxisZ               : FB_Component_BasicAxis := (Name := 'AxisZ');
	AxisQ               : FB_Component_BasicAxis := (Name := 'AxisQ Tangential'); 
	
	
	NciChannel          	: FB_NciChannel := (Name := 'NCI Channel 1');
	NciChannelTangential	: FB_NciChannelTangential := (Name := 'NCI Channel Tangential');
	
	
	
	// [Typ osi: 1=X, 2=Y, 3=Z] , [Typ profilu z Enuma]
	ProfilesX : ARRAY[E_MachineProfile.eProduction..E_MachineProfile.eManual] OF ST_AxisProfile;
	ProfilesY : ARRAY[E_MachineProfile.eProduction..E_MachineProfile.eManual] OF ST_AxisProfile;
	ProfilesZ : ARRAY[E_MachineProfile.eProduction..E_MachineProfile.eManual] OF ST_AxisProfile;
	ProfilesQ : ARRAY[E_MachineProfile.eProduction..E_MachineProfile.eManual] OF ST_AxisProfile;
	
	// Flagi określające typ napędu dla konkretnej osi (TRUE = SoE/AX5000, FALSE = CoE)
    AxisX_IsSoE : BOOL := FALSE;
    AxisY_IsSoE : BOOL := FALSE;
    AxisZ_IsSoE : BOOL := FALSE;
 
	CylinderCuttingX : FB_Cylinder := (Name := 'Cylinder X');
    CylinderCuttingY : FB_Cylinder := (Name := 'Cylinder Y');

    // =========================================================
    //  HOMING STRATEGIES
    // =========================================================
    fbHomeStratX        : FB_Homing_StandardNC;
    fbHomeStratY        : FB_Homing_StandardNC;
    fbHomeStratZ        : FB_Homing_StandardNC;
	fbHomeStratQ 		: FB_Homing_Direct;

    // =========================================================
    //  ALARMS
    // =========================================================
    GantryAlarms        : ARRAY[1..GANTRY_ALARM_COUNT] OF FB_TcAlarm;
	
	ResetStratX : FB_ResetRoutine_SoEDrive;
	ResetStratY : FB_ResetRoutine_SoEDrive;
	ResetStratZ : FB_ResetRoutine_SoEDrive;

END_VAR

VAR CONSTANT
    GANTRY_ALARM_COUNT  : INT := 5;
END_VAR

METHOD PROTECTED Aborting
VAR
    i               : UDINT;
    SubModulesReady : BOOL := TRUE;
END_VAR
VAR_INST
    AbortStepTimer  : TON; 
END_VAR
CASE _CurrentMode OF

//=================================PRODUCTION MODE==================================
// POUs/GantryXYZ/FB_GantryXYZ.TcPOU -> Metoda Aborting

E_PMLUnitMode.ePMLUnitMode_Production:
    CASE SequenceState OF
        0:
            NoStateTasksToComplete := FALSE;
            
            // Logujemy rozpoczęcie procedury Abort
            ADSLOGSTR(ADSLOG_MSGTYPE_HINT, 'Aborting [0]: Zatrzymywanie kanałów i resetowanie błędów NCI...', '');
            
            NciChannel.Stop();
            NciChannelTangential.Stop();
            
            NciChannel.ResetChannel();
            NciChannelTangential.ResetChannel(); 

            AbortStepTimer(IN:=FALSE);
            SequenceState := 10;

        10:
            AbortStepTimer(IN:=TRUE, PT:=T#300MS); 
            IF AbortStepTimer.Q THEN
                AbortStepTimer(IN:=FALSE);
                
                ADSLOGSTR(ADSLOG_MSGTYPE_HINT, 'Aborting [10]: Nakazano rozpięcie (Ungroup) grup 4 i 5.', '');
                
                NciChannel.Ungroup();
                NciChannelTangential.Ungroup(); 
                SequenceState := 20;
            END_IF

        20:
            // Sprawdzanie warunku z logowaniem co jakiś czas (jeśli utknie)
            IF NOT NciChannel.IsGrouped AND NOT NciChannelTangential.IsGrouped THEN
                
                ADSLOGSTR(ADSLOG_MSGTYPE_HINT, 'Aborting [20]: Grupy rozpięte. Wyłączanie napędów i zwalnianie executorów.', '');

                AxisX.Disable();
                AxisY.Disable();
                AxisZ.Disable();
                AxisQ.Disable(); 
        
                IO.SpindleEnable := FALSE;
                IO.CoolingEnable := FALSE;
                
                CylinderCuttingX.Retract();
                CylinderCuttingY.Retract();
        
                fbHomeStratX.Abort();
                fbHomeStratY.Abort();
                fbHomeStratZ.Abort();
				fbHomeStratQ.Abort();
                
                ExecutorCutX.Abort();
                ExecutorCutY.Abort();
                ExecutorGrooveXY.Abort();
                ExecutorNCI.Abort();
                ExecTangentialFeed.Abort();
				ExecutorDrill.Abort();
                
                SequenceState := 30;
            END_IF
    
        30:
            ADSLOGSTR(ADSLOG_MSGTYPE_HINT, 'Aborting [30]: Procedura Abort zakończona sukcesem.', '');
            StateTasksComplete := TRUE;
            
    END_CASE

	//=================================MAINTENANCE & MANUAL MODE==================================
	E_PMLUnitMode.ePMLUnitMode_Maintenance, E_PMLUnitMode.ePMLUnitMode_Manual:

	CASE SequenceState OF
    
		0:
			NoStateTasksToComplete := FALSE;
			SequenceState          := SequenceState + 10;
		
		10:
			AxisX.Disable();
			AxisY.Disable();
			AxisZ.Disable();
			
			CylinderCuttingX.Retract();
			CylinderCuttingY.Retract();
			
			IO.CoolingEnable := FALSE;
			IO.SpindleEnable := FALSE;
	
			SequenceState := SequenceState + 10;
		
		20:
			StateTasksComplete := TRUE;

	END_CASE
	
END_CASE

SUPER^.Aborting();
END_METHOD

//Homing always uses Acc, Decc, Jerk directly from the Parameters. Default Acc, Default Decc, Default Jerk for each axis.
METHOD ApplyProfile
VAR_INPUT
    RequestedProfile : E_MachineProfile;
END_VAR

AxisX.WriteParameter(MC_AxisParameter.AxisMinSoftPosLimit, ProfilesX[RequestedProfile].SoftLimitMin);
AxisX.WriteParameter(MC_AxisParameter.AxisMaxSoftPosLimit, ProfilesX[RequestedProfile].SoftLimitMax);
AxisX.Acceleration := ProfilesX[RequestedProfile].Acceleration;
AxisX.Deceleration := ProfilesX[RequestedProfile].Deceleration;
AxisX.Jerk         := ProfilesX[RequestedProfile].Jerk;

AxisY.WriteParameter(MC_AxisParameter.AxisMinSoftPosLimit, ProfilesY[RequestedProfile].SoftLimitMin);
AxisY.WriteParameter(MC_AxisParameter.AxisMaxSoftPosLimit, ProfilesY[RequestedProfile].SoftLimitMax);
AxisY.Acceleration := ProfilesY[RequestedProfile].Acceleration;
AxisY.Deceleration := ProfilesY[RequestedProfile].Deceleration;
AxisY.Jerk         := ProfilesY[RequestedProfile].Jerk;

AxisZ.WriteParameter(MC_AxisParameter.AxisMinSoftPosLimit, ProfilesZ[RequestedProfile].SoftLimitMin);
AxisZ.WriteParameter(MC_AxisParameter.AxisMaxSoftPosLimit, ProfilesZ[RequestedProfile].SoftLimitMax);
AxisZ.Acceleration := ProfilesZ[RequestedProfile].Acceleration;
AxisZ.Deceleration := ProfilesZ[RequestedProfile].Deceleration;
AxisZ.Jerk         := ProfilesZ[RequestedProfile].Jerk;

AxisQ.WriteParameter(MC_AxisParameter.AxisMinSoftPosLimit, ProfilesQ[RequestedProfile].SoftLimitMin);
AxisQ.WriteParameter(MC_AxisParameter.AxisMaxSoftPosLimit, ProfilesQ[RequestedProfile].SoftLimitMax);
AxisQ.Acceleration := ProfilesQ[RequestedProfile].Acceleration;
AxisQ.Deceleration := ProfilesQ[RequestedProfile].Deceleration;
AxisQ.Jerk         := ProfilesQ[RequestedProfile].Jerk;
AxisQ.Velocity	   := ProfilesQ[RequestedProfile].Velocity;
END_METHOD

METHOD PROTECTED Clearing
VAR
	i				: UDINT;
	SubModulesReady : BOOL := TRUE;
END_VAR
VAR_INST
    LogTimer        : TON; // Timer do opóźniania logów, żeby nie zaspamować konsoli
END_VAR
CASE SequenceState OF
    0:
        NoStateTasksToComplete := FALSE;
        SequenceState          := SequenceState + 10;
    10:
		AxisX.Reset();
		AxisY.Reset();
		AxisZ.Reset();
        AxisQ.Reset(); 
		AxisX.Axis.PlcToNc.ExtSetPos := 2;
		AxisY.Axis.PlcToNc.ExtSetPos := 2;
		
        
        NciChannel.ResetChannel();
        NciChannelTangential.ResetChannel();

		SequenceState := SequenceState + 10;
		
    20:
        StateTasksComplete := TRUE;
END_CASE

SUPER^.Clearing();


LogTimer(IN := (SequenceState = 20), PT := T#2S);

IF LogTimer.Q THEN
    LogTimer(IN := FALSE); 
    
    IF AxisQ.Error THEN
        ADSLOGDINT(ADSLOG_MSGTYPE_ERROR, 'CLEARING BLOCKED BY: AxisQ! ErrorID: %d', UDINT_TO_DINT(AxisQ.ErrorID));
    END_IF
    
    IF NciChannelTangential.ChannelError THEN
        ADSLOGDINT(ADSLOG_MSGTYPE_ERROR, 'CLEARING BLOCKED BY: NciChannelTangential! ErrorID: %d', UDINT_TO_DINT(NciChannelTangential.ChannelErrorId));
    END_IF
    
    IF NciChannel.ChannelError THEN
        ADSLOGDINT(ADSLOG_MSGTYPE_ERROR, 'CLEARING BLOCKED BY: NciChannel! ErrorID: %d', UDINT_TO_DINT(NciChannel.ChannelErrorId));
    END_IF
END_IF
END_METHOD

PROPERTY Config : ST_GantryXYZ_Config
GET
Config := GantryXYZ_HMI.Config;
END_GET
SET
GantryXYZ_HMI.Config.CutterXOffsetX   := LIMIT(_Limits.CutterXOffsetX.MinVal, Config.CutterXOffsetX, _Limits.CutterXOffsetX.MaxVal);
GantryXYZ_HMI.Config.CutterXOffsetY   := LIMIT(_Limits.CutterXOffsetY.MinVal, Config.CutterXOffsetY, _Limits.CutterXOffsetY.MaxVal);
GantryXYZ_HMI.Config.CutterYOffsetX   := LIMIT(_Limits.CutterYOffsetX.MinVal, Config.CutterYOffsetX, _Limits.CutterYOffsetX.MaxVal);
GantryXYZ_HMI.Config.CutterYOffsetY   := LIMIT(_Limits.CutterYOffsetY.MinVal, Config.CutterYOffsetY, _Limits.CutterYOffsetY.MaxVal);
GantryXYZ_HMI.Config.CuttingSpeedXY  := LIMIT(_Limits.CuttingSpeedXY.MinVal, Config.CuttingSpeedXY, _Limits.CuttingSpeedXY.MaxVal);

GantryXYZ_HMI.Config.GroovingSpeedXY := LIMIT(_Limits.GroovingSpeedXY.MinVal, Config.GroovingSpeedXY, _Limits.GroovingSpeedXY.MaxVal);
GantryXYZ_HMI.Config.GroovingSpeedZ  := LIMIT(_Limits.GroovingSpeedZ.MinVal, Config.GroovingSpeedZ, _Limits.GroovingSpeedZ.MaxVal);
GantryXYZ_HMI.Config.GroovingSpeedZ   := LIMIT(_Limits.GroovingSpeedZ.MinVal, Config.GroovingSpeedZ, _Limits.GroovingSpeedZ.MaxVal);

GantryXYZ_HMI.Config.RapidSpeedX      := LIMIT(_Limits.RapidSpeedX.MinVal, Config.RapidSpeedX, _Limits.RapidSpeedX.MaxVal);
GantryXYZ_HMI.Config.RapidSpeedY      := LIMIT(_Limits.RapidSpeedY.MinVal, Config.RapidSpeedY, _Limits.RapidSpeedY.MaxVal);
GantryXYZ_HMI.Config.RapidSpeedZ      := LIMIT(_Limits.RapidSpeedZ.MinVal, Config.RapidSpeedZ, _Limits.RapidSpeedZ.MaxVal);

GantryXYZ_HMI.Config.CuttingIdleTime  := LIMIT(_Limits.CuttingIdleTime.MinVal, Config.CuttingIdleTime, _Limits.CuttingIdleTime.MaxVal);
GantryXYZ_HMI.Config.GroovingIdleTime := LIMIT(_Limits.GroovingIdleTime.MinVal, Config.GroovingIdleTime, _Limits.GroovingIdleTime.MaxVal);

GantryXYZ_HMI.Config.GlobalOffsetX := LIMIT(_Limits.GlobalOffsetX.MinVal, Config.GlobalOffsetX, _Limits.GlobalOffsetX.MaxVal);
GantryXYZ_HMI.Config.GlobalOffsetY := LIMIT(_Limits.GlobalOffsetY.MinVal, Config.GlobalOffsetY, _Limits.GlobalOffsetY.MaxVal);
GantryXYZ_HMI.Config.GlobalOffsetZ := LIMIT(_Limits.GlobalOffsetZ.MinVal, Config.GlobalOffsetZ, _Limits.GlobalOffsetZ.MaxVal);
GantryXYZ_HMI.Config.RawBoardX     := LIMIT(_Limits.RawBoardX.MinVal, Config.RawBoardX, _Limits.RawBoardX.MaxVal);
GantryXYZ_HMI.Config.RawBoardY     := LIMIT(_Limits.RawBoardY.MinVal, Config.RawBoardY, _Limits.RawBoardY.MaxVal);
GantryXYZ_HMI.Config.RawBoardZ      := LIMIT(_Limits.RawBoardZ.MinVal, Config.RawBoardZ, _Limits.RawBoardZ.MaxVal);
GantryXYZ_HMI.Config.SafeClearanceZ := LIMIT(_Limits.SafeClearanceZ.MinVal, Config.SafeClearanceZ, _Limits.SafeClearanceZ.MaxVal);

GantryXYZ_HMI.Config.RapidSpeedQ := LIMIT(_Limits.RapidSpeedQ.MinVal, Config.RapidSpeedQ, _Limits.RapidSpeedQ.MaxVal);

GantryXYZ_HMI.Config.AxisQ_SavedPos := Config.AxisQ_SavedPos;
END_SET
END_PROPERTY

METHOD PROTECTED CreateEvents
VAR_INPUT
END_VAR
// Add your event creation here
F_CreateAllEventsInClass(Alarms     := GantryAlarms,
                         ClassSize  := SIZEOF(TC_EVENTS.Gantry),
                         pInitEvent := ADR(TC_EVENTS.Gantry.InitReferenceEvent),
                         Prefix     := _Name);

// Super call to base
SUPER^.CreateEvents();
END_METHOD

METHOD CyclicLogic
VAR_INPUT
END_VAR
IF NOT _InitComplete THEN
    _InitComplete := Initialize();
    RETURN;
END_IF

SUPER^.CyclicLogic();

fbHomeStratX.bSensorInput := IO.ProximitySensorX;
fbHomeStratY.bSensorInput := IO.ProximitySensorY;
fbHomeStratZ.bSensorInput := IO.ProximitySensorZ;

fbHomeStratX.RapidVelocity := GantryXYZ_HMI.Config.RapidSpeedX;
fbHomeStratY.RapidVelocity := GantryXYZ_HMI.Config.RapidSpeedY;

fbHomeStratZ.RapidVelocity := GantryXYZ_HMI.Config.RapidSpeedZ;
//Axis Z needs to be homed always, because doesn't have an encoder 
fbHomeStratZ.bForceHoming := TRUE;

fbHomeStratX.CyclicLogic();
fbHomeStratY.CyclicLogic();
fbHomeStratZ.CyclicLogic();
fbHomeStratQ.CyclicLogic();

NciChannel.CyclicLogic();

ExecutorCutX.CyclicLogic();
ExecutorCutY.CyclicLogic();
ExecutorGrooveXY.CyclicLogic();
ExecutorNCI.CyclicLogic();
ExecTangentialFeed.CyclicLogic();
ExecutorDrill.CyclicLogic();

//Set the current alarm severity for this module
_CurrentAlarmSeverity := F_GetMaxSeverityRaised(Alarms := GantryAlarms, CurrentSeverity := _CurrentAlarmSeverity);

// Śledzenie i zapamiętywanie pozycji osi Q dla noża tangencjalnego
IF AxisQ.Axis.Status.Homed THEN 
    GantryXYZ_HMI.Config.AxisQ_SavedPos := AxisQ.Axis.NcToPlc.ActPos;
//	fbHomeStratQ.ReferencePosition := GantryXYZ_HMI.Config.AxisQ_SavedPos;
END_IF
END_METHOD

METHOD PROTECTED Execute
VAR
    localConfig : ST_RecipeBuilder_Config; // Zmienna pomocnicza dla kompilatora
END_VAR
CASE _CurrentMode OF

    //=================================PRODUCTION MODE==================================
    E_PMLUnitMode.ePMLUnitMode_Production:
        CASE SequenceState OF
            0:
                NoStateTasksToComplete := FALSE;
                // LOG: Start sekwencji
                ADSLOGSTR(ADSLOG_MSGTYPE_HINT, 'MainSeq: Rozpoczynam nowa sekwencje produkcyjna', '');
                SequenceState := 10;
                
            10: 
                SequenceState := 20;
                
			20: 
				IF _RecipeBuilder <> 0 THEN
					
					// Zależność dla FeedTable
					IF _RecipeBuilder.ExecutionRoute = E_ExecutionRoute.eFeedTable THEN
						_RecipeBuilder.GeometryWriter := ExecTangentialFeed;
					END_IF
					
					// 1. PO PROSTU KAZEMY RECEPCIE PRACOWAĆ (nie sprawdzamy co zwraca funkcja!)
					_RecipeBuilder.Build();
					
					// 2. SPRAWDZAMY FLAGI STANU
					IF _RecipeBuilder.Done THEN 
						
						// ========================================================
						// SUKCES - ROZWIDLENIE DLA FAZY 1
						// ========================================================
						localConfig := _RecipeBuilder.Config;
						
						CASE _RecipeBuilder.ExecutionRoute OF
							E_ExecutionRoute.ePTP:
								ADSLOGSTR(ADSLOG_MSGTYPE_HINT, 'MainSeq: Start Fazy 1 - Tryb PTP', '');
								SequenceState := 30; 
								
							E_ExecutionRoute.eGCode:
								ADSLOGSTR(ADSLOG_MSGTYPE_HINT, 'MainSeq: Start Fazy 1 - Tryb G-Code', '');
								SequenceState := 40;                             
								
							E_ExecutionRoute.eFeedTable:
								ADSLOGSTR(ADSLOG_MSGTYPE_HINT, 'MainSeq: Start Fazy 1 - Tryb FeedTable', '');
								SequenceState := 60; 
						END_CASE
						
					ELSIF _RecipeBuilder.Error THEN
						
						// ========================================================
						// PORAŻKA 
						// ========================================================
						ADSLOGSTR(ADSLOG_MSGTYPE_ERROR, 'MainSeq: Krok 20 - Recepta zglosila ERROR!', '');
						RaiseAlarmWithStrings(GantryAlarms[1], 'Blad budowania recepty! Sprawdz wymiary z HMI.', '');
						ChangeState(E_PMLCommand.ePMLCommand_Abort);
						SequenceState := 999;
			
					END_IF
					// Jeśli nie jest ani Done, ani Error, to maszyna po prostu nic nie robi 
					// i przechodzi do następnego cyklu PLC, dając recepcie czas na pracę (bo flaga _Busy jest aktywna).
			
				ELSE
					// Brak buildera = zły numer programu
					ADSLOGSTR(ADSLOG_MSGTYPE_ERROR, 'MainSeq: BLAD KRYTYCZNY! Brak obiektu _RecipeBuilder.', '');
					ChangeState(E_PMLCommand.ePMLCommand_Abort);
					SequenceState := 999;
				END_IF

            // ========================================================
            // FAZA 1: NARZĘDZIE GŁÓWNE
            // ========================================================
            
            // --- 1A: Wykonanie w trybie PTP (np. GrooveXY) ---
            30: 
                IF ExecutorGrooveXY.Execute() THEN SequenceState := 35; END_IF
            35: 
                IF ExecutorGrooveXY.Done THEN 
                    SequenceState := 70; 
                ELSIF ExecutorGrooveXY.Error THEN
                    RaiseAlarmWithStrings(GantryAlarms[1], 'Blad w Executorze PTP', '');
                    ChangeState(E_PMLCommand.ePMLCommand_Abort);
                    SequenceState := 999;
                END_IF
                
            // --- 1B: Wykonanie w trybie G-Code ---
            40:
                IF ExecutorNCI.Execute() THEN SequenceState := 45; END_IF
            45:
                IF ExecutorNCI.Done THEN 
                    SequenceState := 70;
                ELSIF ExecutorNCI.Error THEN
                    RaiseAlarmWithStrings(GantryAlarms[1], 'Krytyczny Blad NCI G-Code', '');
                    ChangeState(E_PMLCommand.ePMLCommand_Abort);
                    SequenceState := 999; 
                END_IF
                
            // --- 1C: Wykonanie w trybie FeedTable ---
            60:
                IF ExecTangentialFeed.Execute() THEN SequenceState := 65; END_IF
            65:
                IF ExecTangentialFeed.Done THEN 
                    SequenceState := 70;
                ELSIF ExecTangentialFeed.Error THEN
                    RaiseAlarmWithStrings(GantryAlarms[1], 'Krytyczny Blad NCI FeedTable', '');
                    ChangeState(E_PMLCommand.ePMLCommand_Abort);
                    SequenceState := 999; 
                END_IF

				
			// ========================================================
			// FAZA 1.5: WIERCENIE OTWORÓW (Opcjonalne dla każdej recepty)
			// ========================================================
			70:
				IF ExecutorDrill.Execute() THEN 
					ADSLOGSTR(ADSLOG_MSGTYPE_HINT, 'MainSeq: Faza 1.5 - Start operacji wiercenia otworów', '');
					SequenceState := 75;
				END_IF
			75:
				IF ExecutorDrill.Done THEN 
					SequenceState := 100; // Sukces -> Przejście do Fazy 2 (Docinki pneumatyczne)
				ELSIF ExecutorDrill.Error THEN
					RaiseAlarmWithStrings(GantryAlarms[1], 'Krytyczny Blad Executora Wiercenia', '');
					ChangeState(E_PMLCommand.ePMLCommand_Abort);
					SequenceState := 999; 
				END_IF	
				
				

            // ========================================================
            // FAZA 2: DOCINKA PNEUMATYCZNA (Wspólna dla wszystkich)
            // ========================================================
            100: 
                IF ExecutorCutY.Execute() THEN 
                    ADSLOGSTR(ADSLOG_MSGTYPE_HINT, 'MainSeq: Faza 2 - Start operacji CutY', '');
                    SequenceState := 110; 
                END_IF
            110: 
                IF ExecutorCutY.Done THEN 
                    SequenceState := 120;
                ELSIF ExecutorCutY.Error THEN
                    RaiseAlarmWithStrings(GantryAlarms[1], 'Blad w CutY', '');
                    ChangeState(E_PMLCommand.ePMLCommand_Abort);
                    SequenceState := 999;
                END_IF
                
            120: 
                IF ExecutorCutX.Execute() THEN 
                    ADSLOGSTR(ADSLOG_MSGTYPE_HINT, 'MainSeq: Faza 2 - Start operacji CutX', '');
                    SequenceState := 130; 
                END_IF
            130: 
                IF ExecutorCutX.Done THEN 
                    SequenceState := 1000; // Koniec całego detalu!
                ELSIF ExecutorCutX.Error THEN
                    RaiseAlarmWithStrings(GantryAlarms[1], 'Blad w CutX', '');
                    ChangeState(E_PMLCommand.ePMLCommand_Abort);
                    SequenceState := 999;
                END_IF

            // ========================================================
            // MARTWY KROK DLA BŁĘDÓW
            // ========================================================
            999:
                // Maszyna po prostu tu czeka.
                // W tle PackML przetworzy komendę ChangeState i brutalnie przerwie
                // metodę Execute(), przeskakując do metody Aborting()!
                ;
    
            // ========================================================
            // KONIEC OBRÓBKI 
            // ========================================================
            1000:            
                ADSLOGSTR(ADSLOG_MSGTYPE_HINT, 'MainSeq: Sekwencja produkcyjna zakonczona sukcesem.', '');
                StateTasksComplete := TRUE;
                StateComplete();

        END_CASE

    //=================================MAINTENANCE & MANUAL MODE==================================
    E_PMLUnitMode.ePMLUnitMode_Maintenance, E_PMLUnitMode.ePMLUnitMode_Manual:
        ;
END_CASE
END_METHOD

METHOD FB_init : BOOL
VAR_INPUT
	bInitRetains : BOOL; // if TRUE, the retain variables are initialized (warm start / cold start)
	bInCopyCode : BOOL;  // if TRUE, the instance afterwards gets moved into the copy code (online change)
END_VAR



// ===============================================================================
// LIMIT COMMITTED FROM HMI
// ===============================================================================
_Limits.CutterXOffsetX.MinVal := -200.0;   _Limits.CutterXOffsetX.MaxVal := 200.0;
_Limits.CutterXOffsetY.MinVal := -200.0;   _Limits.CutterXOffsetY.MaxVal := 200.0;
_Limits.CutterYOffsetX.MinVal := -200.0;   _Limits.CutterYOffsetX.MaxVal := 200.0;
_Limits.CutterYOffsetY.MinVal := -200.0;   _Limits.CutterYOffsetY.MaxVal := 200.0;
_Limits.GlobalOffsetX.MinVal   := -20.0;   _Limits.GlobalOffsetX.MaxVal   := 1000.0;
_Limits.GlobalOffsetY.MinVal   := -20.0;   _Limits.GlobalOffsetY.MaxVal   := 2000.0;
_Limits.GlobalOffsetZ.MinVal   := -5.0;     _Limits.GlobalOffsetZ.MaxVal   := 5.0;
_Limits.CuttingSpeedXY.MinVal  := 1.0;     _Limits.CuttingSpeedXY.MaxVal  := 100.0;
_Limits.GroovingSpeedXY.MinVal := 1.0;     _Limits.GroovingSpeedXY.MaxVal := 100.0;
_Limits.GroovingSpeedZ.MinVal  := 1.0;     _Limits.GroovingSpeedZ.MaxVal  := 100.0;
_Limits.RapidSpeedX.MinVal     := 1.0;     _Limits.RapidSpeedX.MaxVal     := 200.0;
_Limits.RapidSpeedY.MinVal     := 1.0;     _Limits.RapidSpeedY.MaxVal     := 200.0;
_Limits.RapidSpeedZ.MinVal     := 1.0;     _Limits.RapidSpeedZ.MaxVal     := 20.0;
_Limits.CuttingIdleTime.MinVal  := 0.0;    _Limits.CuttingIdleTime.MaxVal  := 10.0;
_Limits.GroovingIdleTime.MinVal := 0.0;    _Limits.GroovingIdleTime.MaxVal := 10.0;
_Limits.RawBoardX.MinVal       := 200.0;   _Limits.RawBoardX.MaxVal       := 1220.0;
_Limits.RawBoardY.MinVal       := 200.0;   _Limits.RawBoardY.MaxVal       := 2440.0;
_Limits.RawBoardZ.MinVal       := 1.0;     _Limits.RawBoardZ.MaxVal       := 18.0;
_Limits.SafeClearanceZ.MinVal  := 1.0;     _Limits.SafeClearanceZ.MaxVal  := 5.0;
_Limits.RapidSpeedQ.MinVal 	   := 360; 	   _Limits.RapidSpeedQ.MaxVal := 2160.0; 


InitProfiles();
END_METHOD

// Provides interlocks for HMI control and updates HMI status information for this module
//Only in this place HMI input can overwrite internal data 
METHOD PROTECTED HMICommunication
// This method is called cyclically by CyclicLogic()
SUPER^.HMICommunication();

_ProgramIdRequested   := GantryXYZ_HMI.Command.ProgramIdRequested;

GantryXYZ_HMI.Limits := _Limits;
THIS^.Config := GantryXYZ_HMI.Config;
END_METHOD

METHOD PROTECTED HMIPermissions
//General Mode Based Monitoring and handling of HMI control
CASE _CurrentMode OF
   
 E_PMLUnitMode.ePMLUnitMode_Production:
        CASE _CurrentState OF
            E_PMLState.ePMLState_Stopped:
				AllowHMIControl(ThisModuleOnly := FALSE);
            E_PMLState.ePMLState_Idle:
				AllowHMIControl(ThisModuleOnly := FALSE);
            E_PMLState.ePMLState_Suspended:
         		AllowHMIControl(ThisModuleOnly := FALSE);
            E_PMLState.ePMLState_Execute:
            	AllowHMIControl(ThisModuleOnly := FALSE); 
            E_PMLState.ePMLState_Aborted:
                AllowHMIControl(ThisModuleOnly := FALSE); 
            E_PMLState.ePMLState_Held:
                AllowHMIControl(ThisModuleOnly := FALSE); 
            E_PMLState.ePMLState_Complete:
          		AllowHMIControl(ThisModuleOnly := FALSE); 
        END_CASE
		
    E_PMLUnitMode.ePMLUnitMode_Manual:
        AllowHMIControl(ThisModuleOnly := FALSE); 
	E_PMLUnitMode.ePMLUnitMode_Maintenance:
        AllowHMIControl(ThisModuleOnly := FALSE); 
END_CASE
END_METHOD

//! @summary Basic module initialization logic
METHOD PROTECTED Initialize : BOOL;
VAR
    i                        : UDINT;
    varInfo                  : __SYSTEM.VAR_INFO;
    AllSubUnitsInitialized   : BOOL := TRUE;
    AllComponentsInitialized : BOOL := TRUE;
END_VAR

//! @description This method is called by <c>CyclicLogic()</c> as required
Initialize := FALSE;
CASE DescendantSequenceState OF
    0:
		RegisterComponent(AxisX);
		RegisterComponent(AxisY);	
		RegisterComponent(AxisZ);
		RegisterComponent(AxisQ);	
		RegisterComponent(CylinderCuttingY);
		RegisterComponent(CylinderCuttingX);
		RegisterComponent(NciChannel);
		RegisterComponent(NciChannelTangential); 
        _LogModeChanges         := FALSE;
        _LogStateChanges        := FALSE;
		
        DescendantSequenceState := DescendantSequenceState + 10;
    10:
		// Wczytanie zapisanej pozycji dla noża tangencjalnego
		fbHomeStratQ.ReferencePosition := GantryXYZ_HMI.Config.AxisQ_SavedPos;
		
		// Przypisanie osi do strategii
		fbHomeStratX.Axis := AxisX;
		fbHomeStratY.Axis := AxisY;
		fbHomeStratZ.Axis := AxisZ;
		fbHomeStratQ.Axis := AxisQ;
		
		// Wstrzyknięcie strategii do osi (Dependency Injection)
		AxisX.HomeMethod := fbHomeStratX;
		AxisY.HomeMethod := fbHomeStratY;
		AxisZ.HomeMethod := fbHomeStratZ;
		AxisQ.HomeMethod := fbHomeStratQ;
		
		// Wstrzykiwanie zależności do Executora Cut X
		ExecutorCutX.CutDirection   := E_CutDirection.eCutX;
		ExecutorCutX.AxisX          := AxisX;
		ExecutorCutX.AxisY          := AxisY;
		ExecutorCutX.AxisZ          := AxisZ;
		ExecutorCutX.Cylinder       := CylinderCuttingX; // Podpinamy siłownik X!
		ExecutorCutX.ConfigProvider := THIS^;
		
		// Wstrzykiwanie zależności do Executora Cut Y 
		ExecutorCutY.CutDirection   := E_CutDirection.eCutY;
		ExecutorCutY.AxisX          := AxisX;
		ExecutorCutY.AxisY          := AxisY;
		ExecutorCutY.AxisZ          := AxisZ;
		ExecutorCutY.Cylinder       := CylinderCuttingY; // Podpinamy siłownik Y!
		ExecutorCutY.ConfigProvider := THIS^;
		
		// Wstrzykiwanie zależności do Executora NCI
		ExecutorNCI.AxisX          := AxisX;
		ExecutorNCI.AxisY          := AxisY;
		ExecutorNCI.AxisZ          := AxisZ;
		ExecutorNCI.AxisQ          := AxisQ;
		ExecutorNCI.NciChannel     := NciChannel; // Twój nowy kanał
		ExecutorNCI.ConfigProvider := THIS^;
		
		// Wstrzykiwanie zależności do ExecTangentialFeed
		ExecTangentialFeed.AxisX          := AxisX;
		ExecTangentialFeed.AxisY          := AxisY;
		ExecTangentialFeed.AxisZ          := AxisZ;
		ExecTangentialFeed.AxisQ 		  := AxisQ;
		ExecTangentialFeed.NciChannel     := NciChannelTangential; 
		ExecTangentialFeed.ConfigProvider := THIS^;
		
		// Wstrzykiwanie zależności do Executora Drill PTP
		ExecutorDrill.AxisX := AxisX;
		ExecutorDrill.AxisY := AxisY;
		ExecutorDrill.AxisZ := AxisZ;
		ExecutorDrill.AxisQ := AxisQ;
		ExecutorDrill.ConfigProvider := THIS^;

		// Wstrzyknięcie strategii resetu sprzętowego
		// Oś X
		IF AxisX_IsSoE THEN
			AxisX.ResetMethod := ResetStratX;
		END_IF
		
		// Oś Y
		IF AxisY_IsSoE THEN
			AxisY.ResetMethod := ResetStratY;
		END_IF
		
		// Oś Z
		IF AxisZ_IsSoE THEN
			AxisZ.ResetMethod := ResetStratZ;
		END_IF
			
		// Wstrzykiwanie zależności do Executora Groove XY
		ExecutorGrooveXY.AxisX         := AxisX;
		ExecutorGrooveXY.AxisY         := AxisY;
		ExecutorGrooveXY.AxisZ         := AxisZ;
		ExecutorGrooveXY.ConfigProvider := THIS^;
		
		// Dla zwykłego kanału
		NciChannel.stAxisIds.nX := AxisX.Axis.NcToPlc.AxisId;
		NciChannel.stAxisIds.nY := AxisY.Axis.NcToPlc.AxisId;
		NciChannel.stAxisIds.nZ := AxisZ.Axis.NcToPlc.AxisId;
		NciChannel.stAxisIds.nQ1 := AxisQ.Axis.NcToPlc.AxisId;

		// Dla kanału tangencjalnego 
		NciChannelTangential.stAxisIds.nX  := AxisX.Axis.NcToPlc.AxisId;
		NciChannelTangential.stAxisIds.nY  := AxisY.Axis.NcToPlc.AxisId;
		NciChannelTangential.stAxisIds.nZ  := 0;
		NciChannelTangential.stAxisIds.nQ1 := AxisQ.Axis.NcToPlc.AxisId;
		
        DescendantSequenceState := DescendantSequenceState + 10;
		//initialize persistent

    20:
        //Copy Mode names
        FOR i := 1 TO 3 DO
            ModeNames[i] := F_UnitModeToString(UDINT_TO_DINT(i));
        END_FOR

        DescendantSequenceState := DescendantSequenceState + 10;
    30:
        //Call the Super
        IF SUPER^.Initialize() THEN
			ReadAxisParameters();
            DescendantSequenceState := DescendantSequenceState + 10;
        END_IF
    40:
        Initialize := TRUE;
END_CASE
END_METHOD

METHOD PRIVATE InitProfiles
VAR_INPUT
END_VAR

// ========================
// PROFILE 2: PRODUCTION
// ========================
// --- OŚ X ---
ProfilesX[E_MachineProfile.eProduction].SoftLimitMin := -20.0;
ProfilesX[E_MachineProfile.eProduction].SoftLimitMax := 1200.0;
ProfilesX[E_MachineProfile.eProduction].Acceleration := 1000.0;
ProfilesX[E_MachineProfile.eProduction].Deceleration := 1000.0;
ProfilesX[E_MachineProfile.eProduction].Jerk         := 2000.0;

// --- OŚ Y ---
ProfilesY[E_MachineProfile.eProduction].SoftLimitMin := -20.0;
ProfilesY[E_MachineProfile.eProduction].SoftLimitMax := 2200.0;
ProfilesY[E_MachineProfile.eProduction].Acceleration := 1000.0;
ProfilesY[E_MachineProfile.eProduction].Deceleration := 1000.0;
ProfilesY[E_MachineProfile.eProduction].Jerk         := 2000.0;

// --- OŚ Z ---
ProfilesZ[E_MachineProfile.eProduction].SoftLimitMin := -10.0;
ProfilesZ[E_MachineProfile.eProduction].SoftLimitMax := 90.0;
ProfilesZ[E_MachineProfile.eProduction].Acceleration := 10.0;
ProfilesZ[E_MachineProfile.eProduction].Deceleration := 10.0;
ProfilesZ[E_MachineProfile.eProduction].Jerk         := 50.0;

// --- OŚ Q ---
ProfilesQ[E_MachineProfile.eProduction].SoftLimitMin := -3600.0;
ProfilesQ[E_MachineProfile.eProduction].SoftLimitMax := 3600.0;
ProfilesQ[E_MachineProfile.eProduction].Acceleration := 5000.0;
ProfilesQ[E_MachineProfile.eProduction].Deceleration := 5000.0;
ProfilesQ[E_MachineProfile.eProduction].Jerk         := 10000.0;

// ==================
// PROFIL 3: MANUAL 
// ==================
// --- OŚ X ---
ProfilesX[E_MachineProfile.eManual].SoftLimitMin := -50.0;
ProfilesX[E_MachineProfile.eManual].SoftLimitMax := 1250.0;
ProfilesX[E_MachineProfile.eManual].Acceleration := 1000.0;
ProfilesX[E_MachineProfile.eManual].Deceleration := 1000.0;  
ProfilesX[E_MachineProfile.eManual].Jerk         := 2000.0;

// --- OŚ Y ---
ProfilesY[E_MachineProfile.eManual].SoftLimitMin := -100.0;
ProfilesY[E_MachineProfile.eManual].SoftLimitMax := 2500.0;
ProfilesY[E_MachineProfile.eManual].Acceleration := 1000.0;
ProfilesY[E_MachineProfile.eManual].Deceleration := 1000.0;
ProfilesY[E_MachineProfile.eManual].Jerk         := 2000.0;

// --- OŚ Z ---
ProfilesZ[E_MachineProfile.eManual].SoftLimitMin := -20.0;
ProfilesZ[E_MachineProfile.eManual].SoftLimitMax := 100.0;
ProfilesZ[E_MachineProfile.eManual].Acceleration := 10.0;
ProfilesZ[E_MachineProfile.eManual].Deceleration := 10.0;
ProfilesZ[E_MachineProfile.eManual].Jerk         := 50.0;

// --- OŚ Q ---
ProfilesQ[E_MachineProfile.eManual].SoftLimitMin := -3600.0;
ProfilesQ[E_MachineProfile.eManual].SoftLimitMax := 3600.0;
ProfilesQ[E_MachineProfile.eManual].Acceleration := 5000.0;
ProfilesQ[E_MachineProfile.eManual].Deceleration := 5000.0;
ProfilesQ[E_MachineProfile.eManual].Jerk         := 10000.0;
END_METHOD

METHOD PRIVATE IsZAboveMaterial : BOOL
VAR_INST
    MaterialTopZ : REAL;
END_VAR
MaterialTopZ := GantryXYZ_HMI.Config.GlobalOffsetZ + GantryXYZ_HMI.Config.RawBoardZ;

IF AxisZ.Axis.NcToPlc.ActPos >= MaterialTopZ THEN
    IsZAboveMaterial := TRUE;
ELSE
    IsZAboveMaterial := FALSE;
END_IF
END_METHOD

// Called one Cycle on State Change
METHOD PROTECTED ModeChanged
VAR_INPUT
END_VAR
SUPER^.ModeChanged();
CASE _CurrentMode OF
    E_PMLUnitMode.ePMLUnitMode_Production:
		ApplyProfile(E_MachineProfile.eProduction);	      
    E_PMLUnitMode.ePMLUnitMode_Manual:
		ApplyProfile(E_MachineProfile.eManual);
END_CASE
END_METHOD

METHOD PRIVATE MoveZToSafePosition
VAR_INST
    MaterialTopZ : REAL;
    SafeZ        : REAL;
    SpeedZ       : LREAL;
END_VAR
MaterialTopZ := GantryXYZ_HMI.Config.GlobalOffsetZ + GantryXYZ_HMI.Config.RawBoardZ;
SafeZ := MaterialTopZ + GantryXYZ_HMI.Config.SafeClearanceZ;

SpeedZ := GantryXYZ_HMI.Config.RapidSpeedZ;

IF SpeedZ <= 0.0 THEN
    IF AxisZ.AxisParameters.fRefVeloSearch > 0.0 THEN
        SpeedZ := (AxisZ.AxisParameters.fRefVeloSearch);
    ELSE
        SpeedZ := 5.0;
    END_IF
END_IF

IF SafeZ <= 0.0 THEN
    SafeZ := AxisZ.AxisParameters.fEncRefPosition; 
END_IF

AxisZ.Velocity := SpeedZ;
AxisZ.MoveAbsolute(SafeZ, 0);
END_METHOD

PROPERTY ProgramIdRequested : E_RecipeID
GET
ProgramIdRequested := _ProgramIdRequested;
END_GET
SET
// Aktualizacja zmiennej wewnętrznej
_ProgramIdRequested := ProgramIdRequested;

// Aktualizacja struktury HMI, aby ramka (Frame) na wizualizacji od razu zareagowała na zmianę
GantryXYZ_HMI.Command.ProgramIdRequested := ProgramIdRequested;
END_SET
END_PROPERTY

METHOD PRIVATE ReadAxisParameters
VAR_INPUT
END_VAR
//We use it to parametrize Homing Strategies directly from the UI
IF AxisQ.AxisParameters.fRefVeloSearch > 0.0 THEN
    fbHomeStratQ.HomingVelocity := AxisQ.AxisParameters.fRefVeloSearch;
ELSE
    fbHomeStratQ.HomingVelocity := 50.0;
END_IF

IF AxisX.AxisParameters.fRefVeloSearch > 0.0 THEN
    fbHomeStratX.HomingVelocity := AxisX.AxisParameters.fRefVeloSearch;
ELSE
    fbHomeStratX.HomingVelocity := 50.0;
END_IF

IF AxisY.AxisParameters.fRefVeloSearch > 0.0 THEN
    fbHomeStratY.HomingVelocity := AxisY.AxisParameters.fRefVeloSearch;
ELSE
    fbHomeStratY.HomingVelocity := 50.0;
END_IF

IF AxisZ.AxisParameters.fRefVeloSearch > 0.0 THEN
    fbHomeStratZ.HomingVelocity := AxisZ.AxisParameters.fRefVeloSearch;
ELSE
    fbHomeStratZ.HomingVelocity := 5.0;
END_IF

fbHomeStratX.ReferencePosition := AxisX.AxisParameters.fEncRefPosition;
fbHomeStratY.ReferencePosition := AxisY.AxisParameters.fEncRefPosition;
fbHomeStratZ.ReferencePosition := AxisZ.AxisParameters.fEncRefPosition;
END_METHOD

PROPERTY RecipeBuilder : I_RecipeBuilder
GET
RecipeBuilder := _RecipeBuilder;
END_GET
SET
_RecipeBuilder := RecipeBuilder;

ExecutorCutX.RecipeBuilder := _RecipeBuilder;
ExecutorCutY.RecipeBuilder := _RecipeBuilder;
ExecutorGrooveXY.RecipeBuilder := _RecipeBuilder;
ExecutorNCI.RecipeBuilder := _RecipeBuilder;
ExecTangentialFeed.RecipeBuilder := _RecipeBuilder;
ExecutorDrill.RecipeBuilder := _RecipeBuilder;
END_SET
END_PROPERTY

PROPERTY RefAxisX : I_BasicAxis
GET
RefAxisX := AxisX;
END_GET
END_PROPERTY

METHOD PROTECTED Resetting
VAR
    i : UDINT;
    SubModulesReady : BOOL := TRUE;
END_VAR
VAR_INST
    DelayTimer : TON;
END_VAR
CASE _CurrentMode OF

    E_PMLUnitMode.ePMLUnitMode_Production:
        CASE SequenceState OF
            0:
                NoStateTasksToComplete := FALSE;
                StateTasksComplete     := FALSE;
                SequenceState          := 10;
				DelayTimer(IN := FALSE);
        
            10:
                AxisX.Enable();
                AxisY.Enable();
                AxisZ.Enable();
                AxisQ.Enable();
                SequenceState := 20;
        
            20:
                IF AxisX.Enabled AND AxisY.Enabled AND AxisZ.Enabled AND AxisQ.Enabled THEN
                    SequenceState := 25;
                END_IF
        
			25:
				IF NOT AxisZ.Busy THEN
					IF AxisZ.Axis.Status.Homed THEN
						IF NOT IsZAboveMaterial() THEN
							MoveZToSafePosition();
							DelayTimer(IN := FALSE);
							SequenceState := 27;
						ELSE
							SequenceState := 30;
						END_IF
					ELSE
						SequenceState := 30;
					END_IF
				END_IF
            27:
                IF AxisZ.InPosition THEN
                    SequenceState := 30;
                ELSIF AxisZ.Error THEN
                    SequenceState := 99;
                END_IF
                
            30:   
                fbHomeStratQ.Execute();
                DelayTimer(IN := TRUE, PT := T#700MS);
                IF DelayTimer.Q THEN
                    DelayTimer(IN := FALSE); 
                    SequenceState := 31;
                END_IF
				
			31:	
				IF fbHomeStratQ.Done THEN
                    SequenceState := 32;
				END_IF	
			
			32: 
		    	fbHomeStratZ.Execute();
                DelayTimer(IN := TRUE, PT := T#700MS);
                IF DelayTimer.Q THEN
                    DelayTimer(IN := FALSE); 
                    SequenceState := 34;
                END_IF

            34:     
				fbHomeStratY.Execute();    
                DelayTimer(IN := TRUE, PT := T#700MS);
                IF DelayTimer.Q THEN
                    DelayTimer(IN := FALSE); 
                    SequenceState := 38;
                END_IF


            38: 
				fbHomeStratX.Execute();    
                DelayTimer(IN := TRUE, PT := T#700MS);
                IF DelayTimer.Q THEN
                    DelayTimer(IN := FALSE); 
                    SequenceState := 44;
                END_IF
				
        
			44: 	
				IF fbHomeStratX.Done AND fbHomeStratY.Done THEN
                    SequenceState := 50;
                ELSIF fbHomeStratX.Error OR fbHomeStratY.Error OR fbHomeStratQ.Error THEN
                    SequenceState := 99;
                END_IF
				
            50:
                StateTasksComplete := TRUE;
                SequenceState      := 0; 
        
            99:
                ChangeState(E_PMLCommand.ePMLCommand_Abort);
                
        END_CASE

    E_PMLUnitMode.ePMLUnitMode_Maintenance, E_PMLUnitMode.ePMLUnitMode_Manual:
        CASE SequenceState OF
            0:
                NoStateTasksToComplete := FALSE;
                SequenceState := 10;

            10:
                AxisX.Enable();
                AxisY.Enable();
                AxisZ.Enable();
                AxisQ.Enable();

                IF AxisX.Enabled AND AxisY.Enabled AND AxisZ.Enabled AND AxisQ.Enabled THEN
                    SequenceState := 20;
                END_IF

            20:
                StateTasksComplete := TRUE;
        END_CASE

END_CASE

SUPER^.Resetting();
END_METHOD

// Called one Cycle on State Change
METHOD PROTECTED StateChanged
VAR_INPUT
END_VAR
SUPER^.StateChanged();

CASE _CurrentMode OF    
//    E_PMLUnitMode.ePMLUnitMode_Production:
//   CASE _CurrentState OF
//            E_PMLState.ePMLState_Resetting:
//            	ApplyProfile(E_MachineProfile.eHoming);
//        	  END_CASE
//    E_PMLUnitMode.ePMLUnitMode_Manual:
//				;
//        END_CASE
//    E_PMLUnitMode.ePMLUnitMode_Maintenance:
//				;   
//        END_CASE
END_CASE
END_METHOD

END_FUNCTION_BLOCK

// ---- POUs/Executor/FB_Exec_Pneumatic_PTP.TcPOU
FUNCTION_BLOCK FB_Exec_Pneumatic_PTP EXTENDS FB_ExecutorBase
VAR
	_CutDirection : E_CutDirection; //   0 - Cutter direction X, 1 - Cutter direction Y, you can add more in the Enum
END_VAR

PROPERTY CutDirection : E_CutDirection
GET
CutDirection := _CutDirection;
END_GET
SET
_CutDirection := CutDirection;
END_SET
END_PROPERTY

METHOD PUBLIC CyclicLogic
VAR_INST
    localConfig   : ST_GantryXYZ_Config;
    currentSeg    : ST_CutSegment;
    
    // Ujednolicone zmienne pomocnicze
    totalSegments : INT;
    offsetX       : REAL;
    offsetY       : REAL;
END_VAR
// --- START LOGIKI ---
StepTimer();

IF _RecipeBuilder = 0 OR _ConfigProvider = 0 THEN RETURN; END_IF

localConfig := _ConfigProvider.Config;

// ========================================================
// MAGICZNY ROZDZIELACZ Z ENUMEM
// ========================================================
CASE CutDirection OF
    E_CutDirection.eCutX:
        IF iCurrentSegment < 1 OR iCurrentSegment > 1000 THEN iCurrentSegment := 1; END_IF
        currentSeg    := _RecipeBuilder.SegmentsCutX[iCurrentSegment];
        totalSegments := _RecipeBuilder.SegmentsToCutX;
        offsetX       := localConfig.CutterXOffsetX;
        offsetY       := localConfig.CutterXOffsetY;
        
    E_CutDirection.eCutY:
        IF iCurrentSegment < 1 OR iCurrentSegment > 1000 THEN iCurrentSegment := 1; END_IF
        currentSeg    := _RecipeBuilder.SegmentsCutY[iCurrentSegment];
        totalSegments := _RecipeBuilder.SegmentsToCutY;
        offsetX       := localConfig.CutterYOffsetX;
        offsetY       := localConfig.CutterYOffsetY;
        
END_CASE
// ========================================================

CASE nStep OF
    0: // IDLE
    
    5: // INIT
        IF _AxisX.Enable() AND _AxisY.Enable() AND _AxisZ.Enable() THEN
            IF totalSegments <= 0 THEN
                //Trace(Message := 'Step 5: Brak segmentow do ciecia. Koniec (1000).');
                nStep := 1000;
                RETURN;
            END_IF;
            
            _AxisX.Velocity := localConfig.RapidSpeedX;
            _AxisY.Velocity := localConfig.RapidSpeedY;
            _AxisZ.Velocity := localConfig.RapidSpeedZ;

            iCurrentSegment := 1;
            IF NOT _AxisX.Busy AND NOT _AxisY.Busy AND NOT _AxisZ.Busy THEN 
                //Trace(Message := CONCAT('Step 5: Start ciecia. Kierunek: ', TO_STRING(CutDirection)));
                nStep := 10; 
            END_IF     
        END_IF

    // -------- Dojazd do początku cięcia --------
    10:
        //Trace(Message := CONCAT('Step 10: Dojazd do START. Segment: ', TO_STRING(iCurrentSegment)));
        //Trace(Message := CONCAT('--- Kopia X: ', TO_STRING(iCurrentCopyX)));
        //Trace(Message := CONCAT('--- Kopia Y: ', TO_STRING(iCurrentCopyY)));
        //Trace(Message := CONCAT('--- Target Start X: ', TO_STRING(currentSeg.Start.X)));
        //Trace(Message := CONCAT('--- Target Start Y: ', TO_STRING(currentSeg.Start.Y)));
        
        MoveToXY(currentSeg.Start.X, currentSeg.Start.Y, offsetX, offsetY);
        nStep := 20;

    20: // Czekamy na pozycję XY
        IF _AxisX.Error OR _AxisY.Error THEN 
            //Trace(Message := 'Step 20: BLAD OSI X LUB Y!');
            nStep := 999; 
        ELSIF _AxisX.InPosition AND _AxisY.InPosition THEN 
            nStep := 30; 
        END_IF

    30: // Wysunięcie siłownika
        //Trace(Message := 'Step 30: Wysuwanie cylindra (Extend)');
        _Cylinder.Extend();
        nStep := 40;

    40: 
        IF _Cylinder.Extended THEN
            //Trace(Message := 'Step 40: Cylinder wysuniety. Ustawianie predkosci roboczej.');
			_AxisX.Velocity := localConfig.CuttingSpeedXY;
            _AxisY.Velocity := localConfig.CuttingSpeedXY;
            nStep := 50;
        ELSIF _Cylinder.Error THEN 
            //Trace(Message := 'Step 40: BLAD CYLINDRA (Wysuw)!');
            nStep := 999; 
        END_IF
            
    50: // Czekanie (Idle Time)
        StepTimer(IN := TRUE, PT := REAL_TO_TIME(localConfig.CuttingIdleTime * 1000.0));
        IF StepTimer.Q THEN 
            StepTimer(IN := FALSE); 
            nStep := 60; 
        END_IF

    60: // Cięcie XY do końca
        //Trace(Message := CONCAT('Step 60: CIECE DO STOP. Segment: ', TO_STRING(iCurrentSegment)));
        //Trace(Message := CONCAT('--- Target Stop X: ', TO_STRING(currentSeg.Stop.X))); // TUTAJ BYL BLAD! Wczesniej bylo Start.X
        //Trace(Message := CONCAT('--- Target Stop Y: ', TO_STRING(currentSeg.Stop.Y))); // TUTAJ BYL BLAD! Wczesniej bylo Start.Y
        
        MoveToXY(currentSeg.Stop.X, currentSeg.Stop.Y, offsetX, offsetY);
        nStep := 70;

    70: // Czekamy na koniec cięcia
        IF _AxisX.Error OR _AxisY.Error THEN 
            //Trace(Message := 'Step 70: BLAD OSI X LUB Y podczas ciecia!');
            nStep := 999; 
        ELSIF _AxisX.InPosition AND _AxisY.InPosition THEN 
            nStep := 80; 
        END_IF

    80: // Chowanie ostrza
        //Trace(Message := 'Step 80: Chowanie cylindra (Retract)');
        _Cylinder.Retract();
        nStep := 85;

    85: 
        IF _Cylinder.Retracted THEN
             iCurrentSegment := iCurrentSegment + 1;
             nStep := 90;
        ELSIF _Cylinder.Error THEN 
            //Trace(Message := 'Step 85: BLAD CYLINDRA (Chowanie)!');
            nStep := 999; 
        END_IF    

    90: // Drugi Idle Time i obsługa Nestingu
        StepTimer(IN := TRUE, PT := REAL_TO_TIME(localConfig.CuttingIdleTime * 1000.0));
        IF StepTimer.Q THEN
            StepTimer(IN := FALSE);
            _AxisX.Velocity := localConfig.RapidSpeedX;
            _AxisY.Velocity := localConfig.RapidSpeedY;
            
            // CZYSTA PĘTLA NESTINGU
            IF iCurrentSegment > totalSegments THEN
                //Trace(Message := CONCAT('Step 90: Zrobiono wszystkie segmenty dla kopii. Calkowicie zakonczone kopie X: ', TO_STRING(iCurrentCopyX)));
                
                iCurrentCopyX := iCurrentCopyX + 1;
                
                IF iCurrentCopyX > _RecipeBuilder.ActualCopiesX THEN
                    iCurrentCopyX := 1;
                    iCurrentCopyY := iCurrentCopyY + 1;
                    
